ACTION actSetupMode:
//***************************************************************
// Implements a jogging based on velocity mode
// Implements homing depending on the axis type
//   Virtual axis: move absolute to 360 degrees
//   Real axis: depending on parameter S-0-0277 ModeHoming or SetAbsRef
//***************************************************************
// Do nothing, when not enabled... 
IF SetupMode.Enable = TRUE THEN
  // Positive edge of Enable ?
  IF NOT bLatchSetupModeEnable THEN
		// SetupMode is only allowed when in ModeAb or ModeAH 
		IF( (AdminCtrlExt._OpMode.en=ModeAH) OR (AdminCtrlExt._OpMode.en=ModeAb) ) THEN
      // store original values 
      rOriVel          := VelModeCtrlExt.Velocity;
      rOriAccel        := VelModeCtrlExt.Acceleration;
      rOriDecel        := AdminCtrlExt.StopDeceleration;  // Defdb00116851 / Defdb00116875  
      rOriPos          := PosModeCtrlExt.Position;
      rOriVelPos       := PosModeCtrlExt.Velocity;
      rOriAccelPos     := PosModeCtrlExt.Acceleration;
      rOriDecelPos     := PosModeCtrlExt.Deceleration;
      enOriAxisMode    := AdminCtrlExt._OpMode.en;
  	  bOriValuesStored := TRUE;
      // activate mode AH *)
      AdminCtrlExt._OpMode.en := ModeAH;
  	  enMyActAxisMode 	      := ModeAH;
  	  uiHomingState 	      := STATE_HOMING_START;
  	  //SetupModeAck.EnableAck  := TRUE; // Acknowledge SetupMode
    ELSE
      // actual not allowed to activate SetupMode
      SUPER^.mSetError( Error      := TRUE, 
                        ErrorID    := RESOURCE_ERROR, 
             	        ErrorIdent := SETUPMODE_OPMODE_ERR);
  	  bOriValuesStored:= FALSE;
    END_IF  
  END_IF // IF NOT bLatchSetupModeEnable THEN
  
  // Check if someone did overwrite our OpMode command?
  IF( (AdminCtrlExt._OpMode.en <> enMyActAxisMode) AND (SetupModeAck.EnableAck = TRUE) ) THEN
    SetupModeAck.EnableAck := FALSE; // remove acknowledge SetupMode
	
  ELSIF SetupMode.Enable = TRUE THEN
  
    //***************************************************************
    // Jogging
    //***************************************************************
    // Jog positive direction 
    IF SetupMode.JogPlus AND NOT SetupMode.JogMinus THEN
      VelModeCtrlExt.Acceleration	:= SetupMode.Accel;
      AdminCtrlExt.StopDeceleration	:= SetupMode.Accel;  // Defdb00116851 / Defdb00116875
      VelModeCtrlExt.Velocity := SetupMode.Vel;
	  AdminCtrlExt._OpMode.en := ModeVel; 
      enMyActAxisMode := ModeVel; 
    	// Jog negative direction 
    ELSIF SetupMode.JogMinus AND NOT SetupMode.JogPlus THEN
      VelModeCtrlExt.Acceleration	:= SetupMode.Accel;
      AdminCtrlExt.StopDeceleration	:= SetupMode.Accel;  // Defdb00116851 / Defdb00116875
      VelModeCtrlExt.Velocity := -SetupMode.Vel;
  	AdminCtrlExt._OpMode.en := ModeVel;  
  	enMyActAxisMode         := ModeVel;
    ELSIF AdminCtrlExt._OpMode.en = ModeVel THEN
      // switch back when coming from Jog (do not disturb homing)
  	AdminCtrlExt._OpMode.en := ModeAH;
  	enMyActAxisMode         := ModeAH;
    END_IF

    //***************************************************************
    // Implements homing depending on the axis type
    // Virtual axis: move absolute to 360 degrees
    // Real axis with closed loop: depending on parameter S-0-0277 ModeHoming or SetAbsRef
    //***************************************************************
  (* Parameter S277 Bit7/6: only read)
				
		7/6	absolute encoder
		x0: absolute encoder not possible (Bit 7 not in use)
		01: absolute encoder is active)
		11: absolute encoder is possible but deactivated *)

    CASE uiHomingState OF
  
    STATE_HOMING_START:		
        // #####################################################################  
      	IF AdminStatusExt.AxisFeatures.OPMODE_POS = FALSE THEN
          uiHomingState := STATE_HOMING_NOT_POSSIBLE; // can not be homed, e.g. open loop
        ELSIF AdminStatusExt.AxisFeatures.REAL_AXIS = TRUE THEN
					uiHomingState := STATE_HOMING_READ_S277;   // continue with read S-0-0277
      	ELSIF AdminStatusExt.AxisFeatures.VIRTUAL_AXIS = TRUE OR AdminStatusExt.AxisFeatures.CONTROLLER_AXIS = TRUE THEN
					uiHomingState := STATE_HOMING_VIRT_AXIS;   // continue with homing virtual axis
      	ELSE 
      	  // undefined axis type
   	  	  SUPER^.mSetError( Error      := TRUE, 
       		                  ErrorID    := RESOURCE_ERROR, 
           		              ErrorIdent := HOMING_CONFIGURATION_ERR);
   	  	  uiHomingState := STATE_HOMING_ERROR;   // continue with error
  		  END_IF
  
    STATE_HOMING_READ_S277:
        // #####################################################################  
      	// first read S-0-0277 when SetupMode is activated
	 			MB_ReadParameterS277(
    		Enable:= TRUE, 
    		ParameterNumber:= FP_S_0_0277, 
    		Axis:= AdminCtrlExt.Axis );
   		  IF MB_ReadParameterS277.Done = TRUE THEN
					// store Value   
					diParameterS277 := MB_ReadParameterS277.Value;
					IF 	(diParameterS277.6 AND NOT diParameterS277.7) OR diParameterS277.8 THEN
		    	  // absolute encoder
						bAbsoluteEncoder := TRUE;
        	  uiHomingState := STATE_HOMING_ABS_REAL_AXIS; // continue with homing an absolute real axis
					ELSE
		    	  // incremental encoder
						bAbsoluteEncoder := FALSE;
        	  uiHomingState := STATE_HOMING_INC_REAL_AXIS; // continue with homing an incremental real axis
					END_IF
					// RESET FB  
    		MB_ReadParameterS277(
       		Enable:= FALSE, 
      		ParameterNumber:= FP_S_0_0277, 
      		Axis:= AdminCtrlExt.Axis );
      	ELSIF MB_ReadParameterS277.Error = TRUE THEN
    		  SUPER^.mSetError( Error      := TRUE, 
                            ErrorID    := MB_ReadParameterS277.ErrorID, 
                            ErrorIdent := MB_ReadParameterS277.ErrorIdent);
					// RESET FB  
    		  MB_ReadParameterS277(
       		  Enable:= FALSE, 
      		  ParameterNumber:= FP_S_0_0277, 
      		  Axis:= AdminCtrlExt.Axis );
        	  uiHomingState := STATE_HOMING_ERROR;   // continue with error
  		  END_IF	// end of 'IF MB_ReadParameterS277.Done = TRUE THEN'		  
	
    STATE_HOMING_ABS_REAL_AXIS:
        // ##################################################################### 
				SetupModeAck.EnableAck  := TRUE; // Acknowledge SetupMode 
    		// Homing for Real-Axis with absolute encoder
      	IF (SetupMode.Homing = TRUE) AND (bHomingOld = FALSE) THEN
       		// Set reference with absolute encoder
       		AdminCtrlExt._OpMode.en := ModeAB;
    			enMyActAxisMode         := ModeAB;
				// wait for Homing finished
      	ELSIF  AdminStatusExt.AbsRefCmdStatus = MB_SERCOS_DATA_END_OK THEN
					// command finished GOOD
					SetupModeAck.HomingAck := TRUE;
					uiHomingState := STATE_HOMING_FINISHED;
					IF SetupMode.Homing = FALSE THEN
		  		  // Input was removed. Switch back to ModeAH. HomingAck stays active for one cycle... 	
		  		  bHomingRemovedBeforeFinished := TRUE;	
					END_IF	
        // Note: problems with IndraDrive Cs. It takes time to switch to AB and the 
        // C0304 "command not allowed in AF" can happen so wait for PowerOff before 
        // setting the command set absolute reference
      	ELSIF (SetupMode.Homing = TRUE) AND 
              (AxisData[AdminCtrlExt.Axis.AxisNo].Axis_Power = FALSE) THEN
       		AdminCtrlExt.SetAbsRef := TRUE;
				ELSIF ( (AdminStatusExt.AbsRefCmdStatus = MB_SERCOS_DATA_INTERRUPTED) OR	
	    	        (AdminStatusExt.AbsRefCmdStatus = MB_SERCOS_DATA_BREAK_ERROR) OR
								(AdminStatusExt.AbsRefCmdStatus = MB_SERCOS_DATA_DATUM_FAULT)    ) THEN
					// command finished BAD
					SetupModeAck.HomingAck := FALSE;
					uiHomingState := STATE_HOMING_FINISHED;
					IF SetupMode.Homing = FALSE THEN
		  		// Input was removed. Switch back to ModeAH. 	
		  		bHomingRemovedBeforeFinished := TRUE;	
					END_IF
        END_IF // end of 'IF (SetupMode.Homing = TRUE) AND (bHomingOld = FALSE) THEN'

    STATE_HOMING_INC_REAL_AXIS:
        // #####################################################################
				SetupModeAck.EnableAck  := TRUE; // Acknowledge SetupMode
    		// Homing for Real-Axis with incremental encoder
      	IF (SetupMode.Homing = TRUE) AND (bHomingOld = FALSE) THEN
       		// Set reference with incremental encoder
       		AdminCtrlExt._OpMode.en := ModeHoming;
    			enMyActAxisMode         := ModeHoming;
      	ELSIF AdminStatusExt.CmdDone THEN
					// wait for Homing finished
					// Homing finished GOOD
					SetupModeAck.HomingAck := TRUE;
					uiHomingState := STATE_HOMING_FINISHED;
					IF SetupMode.Homing = FALSE THEN
		  		// Input was removed. Switch back to ModeAH. HomingAck stays active for one cycle... 	
		  		bHomingRemovedBeforeFinished := TRUE;	
					END_IF
      	ELSIF  DiagStatusExt.Error = TRUE AND SetupMode.Homing = FALSE THEN
					// wait for Homing finished BAD. Stay here untill the Homing is removed
					SetupModeAck.HomingAck := FALSE;
					uiHomingState := STATE_HOMING_FINISHED;
  	    // Input was removed. Switch back to ModeAH. 	
					bHomingRemovedBeforeFinished := TRUE;	
      	END_IF // end of 'IF (SetupMode.Homing = TRUE) AND (bHomingOld = FALSE) THEN'		
   
    STATE_HOMING_VIRT_AXIS:
      // #####################################################################  
			SetupModeAck.EnableAck  := TRUE; // Acknowledge SetupMode
    	// Homing for Virtual-Axis -> Move abs to position 0
      	IF (SetupMode.Homing = TRUE) AND (bHomingOld = FALSE) THEN
					// rising edge on Homing  
    			// Homing for Virtual-Axis: Move to position 0 degrees
					// use SetupMode.Vel and .Accel 
          //PosModeCtrlExt.Velocity 	:= SetupMode.Vel;
          //PosModeCtrlExt.Acceleration := SetupMode.Accel;
          //PosModeCtrlExt.Deceleration := SetupMode.Accel;
					// or set vel and acc to the maximum values 
          PosModeCtrlExt.Velocity 	:= DV_Axis[AdminCtrlExt.Axis.AxisNo].A_0_0032; // or A-0-0033?
          PosModeCtrlExt.Acceleration := DV_Axis[AdminCtrlExt.Axis.AxisNo].A_0_0034-0.001; // - 0,001 to avoid warning
          PosModeCtrlExt.Deceleration := PosModeCtrlExt.Acceleration;
	    	  PosModeCtrlExt.Position 	:= 0.0; 
					AdminCtrlExt._OpMode.en := ModePosAbs;
					enMyActAxisMode         := ModePosAbs;
      	ELSIF  AdminStatusExt.CmdDone AND AdminStatusExt.MODE_POS_ABS THEN
					// wait for Homing finished GOOD
					SetupModeAck.HomingAck := TRUE;
					uiHomingState := STATE_HOMING_FINISHED;
					IF SetupMode.Homing = FALSE THEN
		  		// Input was removed. Switch back to ModeAH. HomingAck stays active for one cycle... 	
		  		bHomingRemovedBeforeFinished := TRUE;	
          END_IF
      	ELSIF  DiagStatusExt.Error = TRUE AND SetupMode.Homing = FALSE THEN
					// wait for Homing finished BAD. Stay here untill the Homing is removed
					SetupModeAck.HomingAck := FALSE;
					uiHomingState := STATE_HOMING_FINISHED;
  	      // Input was removed. Switch back to ModeAH. 	
					bHomingRemovedBeforeFinished := TRUE;	
      	END_IF // end of 'IF (SetupMode.Homing = TRUE) AND (bHomingOld = FALSE) THEN'		
	
  STATE_HOMING_FINISHED:	
        // #####################################################################  
      	IF( ((SetupMode.Homing = FALSE) AND (bHomingOld = TRUE)) OR 
            (bHomingRemovedBeforeFinished = TRUE)                   ) THEN
					// falling edge on Homing or Homing removed before finished, reset to previous settings   
					AdminCtrlExt.SetAbsRef := FALSE;
        	AdminCtrlExt._OpMode.en := ModeAH;
					enMyActAxisMode         := ModeAH;
					// remove Acknowledge
					SetupModeAck.HomingAck := FALSE;
					bHomingRemovedBeforeFinished := FALSE;
					// wait for the next rising edge on Homing input
					IF AdminStatusExt.AxisFeatures.REAL_AXIS = TRUE THEN
						IF bAbsoluteEncoder = TRUE THEN
		      	  // absolute encoder
			  		  uiHomingState := STATE_HOMING_ABS_REAL_AXIS; // continue with homing an absolute real axis
		    	  ELSE
		      	  // incremental encoder
              uiHomingState := STATE_HOMING_INC_REAL_AXIS; // continue with homing an incremental real axis
						END_IF	
          ELSE 
		   		  uiHomingState := STATE_HOMING_VIRT_AXIS;   // continue with homing virtual axis
          END_IF
				END_IF	

    STATE_HOMING_NOT_POSSIBLE:
		  ; // nothing to do
      
    STATE_HOMING_ERROR:
      // #####################################################################  
  		IF AdminCtrlExt.ClearError THEN
     		uiHomingState := STATE_HOMING_START;   // try a new start
  		END_IF	
	   

    ELSE 
        // #####################################################################  
   			// invalid state
   			SUPER^.mSetError( Error      := TRUE, 
       		              ErrorID    := STATE_MACHINE_ERROR, 
          	 	          ErrorIdent := HOMING_STATE_MACHINE_ERR);
   			uiHomingState := STATE_HOMING_ERROR;   // continue with error
	
    END_CASE // end of 'CASE uiHomingState OF'
  END_IF  // end of 'ELSIF SetupModeAck.SetupModeAck = TRUE THEN'
 
// Negative edge of Enable ? AND SetupMode was not aborted by assigning a new OpMode  
ELSIF bLatchSetupModeEnable AND bOriValuesStored = TRUE AND SetupModeAck.EnableAck = TRUE THEN
  // restore original values 
  VelModeCtrlExt.Velocity       := rOriVel;
  VelModeCtrlExt.Acceleration   := rOriAccel;
  AdminCtrlExt.StopDeceleration := rOriDecel;  // Defdb00116851 / Defdb00116875
  PosModeCtrlExt.Position       := rOriPos;
  PosModeCtrlExt.Velocity       := rOriVelPos;
  PosModeCtrlExt.Acceleration   := rOriAccelPos;
  PosModeCtrlExt.Deceleration   := rOriDecelPos;
  AdminCtrlExt._OpMode.en       := enOriAxisMode;
  bOriValuesStored              := FALSE;
  SetupModeAck.EnableAck        := FALSE; // remove acknowledge SetupMode
END_IF // SetupMode.Enable = TRUE

bLatchSetupModeEnable := SetupMode.Enable;
bHomingOld            := SetupMode.Homing;
END_ACTION

ACTION actSyncAccVel:
// Implements writing the Sync-Acceleration into parameter A-0-2791
// and writing the Sync-Velocity into parameter A-0-2790
// ####################################################
// Check if we are in bb. Otherwise we get errors.
// Do this only when sync is supported and the parameters are available.
// Distribute the load with using the axis address
IF AxisData[AdminCtrlExt.Axis.AxisNo].Axis_OperationMode = TRUE    AND 
   AdminStatusExt.AxisFeatures.OPMODE_SYNC = TRUE                   AND 
   (udiCycleCntInP4 > DINT_TO_UDINT(2 * AdminCtrlExt.Axis.AxisNo))     THEN 
  // write SyncAcceleration when changed 
  IF SyncModeCtrlExt.SyncAcceleration <> rLastSyncAcc THEN
    // start transmission 
    SyncModeStatusExt.SyncAccelerationDone := FALSE;
    bExecWrSyncAcc := TRUE;
  END_IF
  IF fbWrSyncAcc.Done = TRUE THEN 
    // finished GOOD transmission 
    SyncModeStatusExt.SyncAccelerationDone := TRUE;
    bExecWrSyncAcc := FALSE;
    // remember old value 
    rLastSyncAcc := SyncModeCtrlExt.SyncAcceleration;
  ELSIF fbWrSyncAcc.Error = TRUE THEN  
    // finished BAD transmission 
    bExecWrSyncAcc := FALSE;
    SUPER^.mSetError( Error      := TRUE, 
                      ErrorID    := fbWrSyncAcc.ErrorID, 
                      ErrorIdent := fbWrSyncAcc.ErrorIdent);
    // remember old value, to not write cyclically bad values 
    rLastSyncAcc := SyncModeCtrlExt.SyncAcceleration;
  END_IF  
  // call FB 
  fbWrSyncAcc(
	Execute:= bExecWrSyncAcc, 
	ParameterNumber:= FP_A_0_2791, 
	Value:= SyncModeCtrlExt.SyncAcceleration, 
	Axis:= AdminCtrlExt.Axis );	
	
  // ####################################################
  // write SyncVelocity when changed 
  IF SyncModeCtrlExt.SyncVelocity <> rLastSyncVel THEN
    // start transmission 
    SyncModeStatusExt.SyncVelocityDone := FALSE;
    bExecWrSyncVel := TRUE;
  END_IF
  IF fbWrSyncVel.Done = TRUE THEN 
    // finished GOOD transmission 
    SyncModeStatusExt.SyncVelocityDone := TRUE;
    bExecWrSyncVel := FALSE;
    // remember old value 
    rLastSyncVel := SyncModeCtrlExt.SyncVelocity;
  ELSIF fbWrSyncVel.Error = TRUE THEN  
    // finished BAD transmission 
    bExecWrSyncVel := FALSE;
    SUPER^.mSetError( Error      := TRUE, 
                      ErrorID    := fbWrSyncVel.ErrorID, 
                      ErrorIdent := fbWrSyncVel.ErrorIdent);
    // remember old value, to not write cyclically bad values 
    rLastSyncVel := SyncModeCtrlExt.SyncVelocity;
  END_IF  
  // call FB 
  fbWrSyncVel(
	Execute:= bExecWrSyncVel, 
	ParameterNumber:= FP_A_0_2790, 
	Value:= SyncModeCtrlExt.SyncVelocity, 
	Axis:= AdminCtrlExt.Axis );	
ELSE
  // reset FBs when not in bb 
  fbWrSyncAcc( Execute:= FALSE,	Axis:= AdminCtrlExt.Axis );	
  fbWrSyncVel( Execute:= FALSE,	Axis:= AdminCtrlExt.Axis );	
END_IF
END_ACTION

ACTION actCopyAxisData_HMI:
// copy AxisData status informations to AxisData_HMI structure to transmit to HMI

AxisData_HMI.dwMotionProfileStatusBits_i    	:=	AxisData[AdminCtrlExt.Axis.AxisNo].dwMotionProfileStatusBits_i;	
AxisData_HMI.FlexProfil_Sync                    :=  AxisData[AdminCtrlExt.Axis.AxisNo].FlexProfil_Sync;                 
AxisData_HMI.FlexProfil_Active                  :=  AxisData[AdminCtrlExt.Axis.AxisNo].FlexProfil_Active;               
AxisData_HMI.FlexProfil_WaitForSwitching        :=  AxisData[AdminCtrlExt.Axis.AxisNo].FlexProfil_WaitForSwitching;     
AxisData_HMI.FlexProfil_Set0_Checked            :=  AxisData[AdminCtrlExt.Axis.AxisNo].FlexProfil_Set0_Checked;         
AxisData_HMI.FlexProfil_Set0_Ok                 :=  AxisData[AdminCtrlExt.Axis.AxisNo].FlexProfil_Set0_Ok;              
AxisData_HMI.FlexProfil_Set1_Checked            :=  AxisData[AdminCtrlExt.Axis.AxisNo].FlexProfil_Set1_Checked;         
AxisData_HMI.FlexProfil_Set1_Ok                 :=  AxisData[AdminCtrlExt.Axis.AxisNo].FlexProfil_Set1_Ok;              
AxisData_HMI.FlexProfil_Set2_Checked            :=  AxisData[AdminCtrlExt.Axis.AxisNo].FlexProfil_Set2_Checked;         
AxisData_HMI.FlexProfil_Set2_Ok                 :=  AxisData[AdminCtrlExt.Axis.AxisNo].FlexProfil_Set2_Ok;              
AxisData_HMI.FlexProfil_Set3_Checked            :=  AxisData[AdminCtrlExt.Axis.AxisNo].FlexProfil_Set3_Checked;         
AxisData_HMI.FlexProfil_Set3_Ok                 :=  AxisData[AdminCtrlExt.Axis.AxisNo].FlexProfil_Set3_Ok;              
AxisData_HMI.FlexProfil_EvtSet0_Checked         :=  AxisData[AdminCtrlExt.Axis.AxisNo].FlexProfil_EvtSet0_Checked;      
AxisData_HMI.FlexProfil_EvtSet0_Ok              :=  AxisData[AdminCtrlExt.Axis.AxisNo].FlexProfil_EvtSet0_Ok;           
AxisData_HMI.FlexProfil_EvtSet1_Checked         :=  AxisData[AdminCtrlExt.Axis.AxisNo].FlexProfil_EvtSet1_Checked;      
AxisData_HMI.FlexProfil_EvtSet1_Ok              :=  AxisData[AdminCtrlExt.Axis.AxisNo].FlexProfil_EvtSet1_Ok;           
AxisData_HMI.FlexProfil_EvtSet2_Checked         :=  AxisData[AdminCtrlExt.Axis.AxisNo].FlexProfil_EvtSet2_Checked;      
AxisData_HMI.FlexProfil_EvtSet2_Ok              :=  AxisData[AdminCtrlExt.Axis.AxisNo].FlexProfil_EvtSet2_Ok;           
AxisData_HMI.FlexProfil_EvtSet3_Checked         :=  AxisData[AdminCtrlExt.Axis.AxisNo].FlexProfil_EvtSet3_Checked;      
AxisData_HMI.FlexProfil_EvtSet3_Ok              :=  AxisData[AdminCtrlExt.Axis.AxisNo].FlexProfil_EvtSet3_Ok;           
AxisData_HMI.dwFlexProfileEventStatusBits_i     :=  AxisData[AdminCtrlExt.Axis.AxisNo].dwFlexProfileEventStatusBits_i; 
AxisData_HMI.Axis_CamTab_0                      :=  AxisData[AdminCtrlExt.Axis.AxisNo].Axis_CamTab_0;                   
AxisData_HMI.Axis_CamTab_1                      :=  AxisData[AdminCtrlExt.Axis.AxisNo].Axis_CamTab_1;                   
AxisData_HMI.Axis_CamTab_2                      :=  AxisData[AdminCtrlExt.Axis.AxisNo].Axis_CamTab_2;                   
AxisData_HMI.Axis_CamSwitching                  :=  AxisData[AdminCtrlExt.Axis.AxisNo].Axis_CamSwitching;               
AxisData_HMI.Axis_InVelocity                    :=  AxisData[AdminCtrlExt.Axis.AxisNo].Axis_InVelocity;                 
AxisData_HMI.Axis_Standstill                    :=  AxisData[AdminCtrlExt.Axis.AxisNo].Axis_Standstill;                 
AxisData_HMI.Axis_InPosition                    :=  AxisData[AdminCtrlExt.Axis.AxisNo].Axis_InPosition;      
AxisData_HMI.Axis_InSynchron                    :=  AxisData[AdminCtrlExt.Axis.AxisNo].Axis_InSynchron;                 
AxisData_HMI.Axis_Warning                       :=  AxisData[AdminCtrlExt.Axis.AxisNo].Axis_Warning;                    
AxisData_HMI.Axis_Error                         :=  AxisData[AdminCtrlExt.Axis.AxisNo].Axis_Error;                      
AxisData_HMI.Axis_Homed                         :=  AxisData[AdminCtrlExt.Axis.AxisNo].Axis_Homed;                      
AxisData_HMI.Axis_InTorque                      :=  AxisData[AdminCtrlExt.Axis.AxisNo].Axis_InTorque;                   
AxisData_HMI.Axis_OperationMode                 :=  AxisData[AdminCtrlExt.Axis.AxisNo].Axis_OperationMode;              
AxisData_HMI.Axis_Inbb                          :=  AxisData[AdminCtrlExt.Axis.AxisNo].Axis_Inbb;                       
AxisData_HMI.Axis_InAb                          :=  AxisData[AdminCtrlExt.Axis.AxisNo].Axis_InAb;                       
AxisData_HMI.Axis_Power                         :=  AxisData[AdminCtrlExt.Axis.AxisNo].Axis_Power;                      
AxisData_HMI.Axis_CmdActive                     :=  AxisData[AdminCtrlExt.Axis.AxisNo].Axis_CmdActive;                  
AxisData_HMI.Axis_ErrInProgress                 :=  AxisData[AdminCtrlExt.Axis.AxisNo].Axis_ErrInProgress;              
AxisData_HMI.Axis_CyclicPosChannelOpen          :=  AxisData[AdminCtrlExt.Axis.AxisNo].Axis_CyclicPosChannelOpen;       
AxisData_HMI.Axis_InMasterPhaseOffset           :=  AxisData[AdminCtrlExt.Axis.AxisNo].Axis_InMasterPhaseOffset;        
AxisData_HMI.Axis_CyclicTrqChannelOpen          :=  AxisData[AdminCtrlExt.Axis.AxisNo].Axis_CyclicTrqChannelOpen;       
AxisData_HMI.Axis_CyclicVelChannelOpen          :=  AxisData[AdminCtrlExt.Axis.AxisNo].Axis_CyclicVelChannelOpen;       
AxisData_HMI.Axis_CyclicAnaChannelOpen          :=  AxisData[AdminCtrlExt.Axis.AxisNo].Axis_CyclicAnaChannelOpen;       
AxisData_HMI.ErrorStop                          :=  AxisData[AdminCtrlExt.Axis.AxisNo].ErrorStop;                       
AxisData_HMI.Stopping                           :=  AxisData[AdminCtrlExt.Axis.AxisNo].Stopping;                        
AxisData_HMI.Homing                             :=  AxisData[AdminCtrlExt.Axis.AxisNo].Homing;                          
AxisData_HMI.PowerOn                            :=  AxisData[AdminCtrlExt.Axis.AxisNo].PowerOn;                         
AxisData_HMI.DiscreteMotion                     :=  AxisData[AdminCtrlExt.Axis.AxisNo].DiscreteMotion;                  
AxisData_HMI.ContinuousMotion                   :=  AxisData[AdminCtrlExt.Axis.AxisNo].ContinuousMotion;                
AxisData_HMI.SynchronizedMotion                 :=  AxisData[AdminCtrlExt.Axis.AxisNo].SynchronizedMotion;              
AxisData_HMI.Standstill                         :=  AxisData[AdminCtrlExt.Axis.AxisNo].Standstill;                      
AxisData_HMI.CoordinatedMotion                  :=  AxisData[AdminCtrlExt.Axis.AxisNo].CoordinatedMotion;               
AxisData_HMI.ControlledMotion                   :=  AxisData[AdminCtrlExt.Axis.AxisNo].ControlledMotion;                
AxisData_HMI.dwAxisCondition_i                  :=  AxisData[AdminCtrlExt.Axis.AxisNo].dwAxisCondition_i;               
AxisData_HMI.rActualPosition_i                  :=  AxisData[AdminCtrlExt.Axis.AxisNo].rActualPosition_i;               
AxisData_HMI.rActualVelocity_i                  :=  AxisData[AdminCtrlExt.Axis.AxisNo].rActualVelocity_i;               
AxisData_HMI.rActualTorqueForce_i               :=  AxisData[AdminCtrlExt.Axis.AxisNo].rActualTorqueForce_i;            
AxisData_HMI.wUserActualDataBitA_i              :=  AxisData[AdminCtrlExt.Axis.AxisNo].wUserActualDataBitA_i;          
AxisData_HMI.wUserActualDataBitB_i              :=  AxisData[AdminCtrlExt.Axis.AxisNo].wUserActualDataBitB_i;          
AxisData_HMI.wUserActualDataBitC_i              :=  AxisData[AdminCtrlExt.Axis.AxisNo].wUserActualDataBitC_i;          
AxisData_HMI.wUserActualDataBitD_i              :=  AxisData[AdminCtrlExt.Axis.AxisNo].wUserActualDataBitD_i;          
AxisData_HMI.dwUserActualDataA_i                :=  AxisData[AdminCtrlExt.Axis.AxisNo].dwUserActualDataA_i;             
AxisData_HMI.dwUserActualDataB_i                :=  AxisData[AdminCtrlExt.Axis.AxisNo].dwUserActualDataB_i;             
AxisData_HMI.dwUserActualDataC_i                :=  AxisData[AdminCtrlExt.Axis.AxisNo].dwUserActualDataC_i;             
AxisData_HMI.dwUserActualDataD_i                :=  AxisData[AdminCtrlExt.Axis.AxisNo].dwUserActualDataD_i;             
AxisData_HMI.dwUserActualDataE_i                :=  AxisData[AdminCtrlExt.Axis.AxisNo].dwUserActualDataE_i;             
AxisData_HMI.dwUserActualDataF_i                :=  AxisData[AdminCtrlExt.Axis.AxisNo].dwUserActualDataF_i;
END_ACTION

METHOD mInitExtension
VAR_INPUT
	index: UINT;
END_VAR
VAR
END_VAR
SUPER^.mInitExtension(index);

IF NOT bFirstInit THEN
	// User: Assigment of user defined axis interface inputs
	SetupMode  REF= arAxisCtrl_gb[index].SetupMode;
	
	// User: Assigment of user defined axis interface outputs
	SetupModeAck REF= arAxisStatus_gb[index].SetupMode;
	AxisData_HMI REF= arAxisStatus_gb[index].AxisData_HMI;
	
	// =================================================================
	// Do not touch the following lines
	// =================================================================
	
	// Set the references for the AxisInterface FB 
	AdminCtrlExt   	REF= arAxisCtrl_gb[index].Admin;
	PosModeCtrlExt    REF= arAxisCtrl_gb[index].PosMode;
	VelModeCtrlExt    REF= arAxisCtrl_gb[index].VelMode;
	SyncModeCtrlExt   REF= arAxisCtrl_gb[index].SyncMode;
	AdminStatusExt    REF= arAxisStatus_gb[index].Admin;
	DiagStatusExt     REF= arAxisStatus_gb[index].Diag;
	PosStatusExt   	REF= arAxisStatus_gb[index].PosMode;
	VelStatusExt      REF= arAxisStatus_gb[index].VelMode;
	SyncModeStatusExt REF= arAxisStatus_gb[index].SyncMode;
	// System: assign references of axis interface refresh FB
	AdminCtrl 				REF= arAxisCtrl_gb[index].Admin;
	PosModeCtrl 			REF= arAxisCtrl_gb[index].PosMode;
	VelModeCtrl 			REF= arAxisCtrl_gb[index].VelMode;
	SyncModeCtrl 			REF= arAxisCtrl_gb[index].SyncMode;
	AdminStatus 			REF= arAxisStatus_gb[index].Admin;
	DiagStatus 				REF= arAxisStatus_gb[index].Diag;
	PosStatus 				REF= arAxisStatus_gb[index].PosMode;
	VelStatus 				REF= arAxisStatus_gb[index].VelMode;
	SyncModeStatus 		REF= arAxisStatus_gb[index].SyncMode;
END_IF
END_METHOD

END_FUNCTION_BLOCK

// IndraMotionMlc1/Application/Utilities/InitAxis
PROGRAM InitAxis
VAR
	index:INT;
END_VAR
VAR_INPUT
	
	arAxisPointer: POINTER TO ARRAY[1..20] OF AXIS_REF;
	uiNUM_FLEXO_F: UINT;
	
END_VAR

FOR index:=1 TO uiNUM_FLEXO_F BY 1 DO
		arAxisCtrl_gb[arAxisPointer^[index].AxisNo].SyncMode.InputRevolution := 1000;
		arAxisCtrl_gb[arAxisPointer^[index].AxisNo].SyncMode.OutputRevolution := 1000;
		arAxisCtrl_gb[arAxisPointer^[index].AxisNo].SyncMode.Master:=VMA_FT1;
		arAxisCtrl_gb[arAxisPointer^[index].AxisNo].SyncMode.StartMode:=RELATIVE;
		arAxisCtrl_gb[arAxisPointer^[index].AxisNo].SyncMode.SyncAcceleration:=1.0;
		arAxisCtrl_gb[arAxisPointer^[index].AxisNo].SyncMode.PhaseOffsetAcc:=1.0;
		arAxisCtrl_gb[arAxisPointer^[index].AxisNo].SyncMode.SyncDirection:=SHORTEST_WAY;
		arAxisCtrl_gb[arAxisPointer^[index].AxisNo].SyncMode.SyncVelocity:=5.0;
	END_FOR

END_PROGRAM

// IndraMotionMlc1/Application/STATE_MACHINE/Winder
PROGRAM Winder
VAR_INPUT
	arAxisPointer: POINTER TO ARRAY[1..20] OF AXIS_REF;
	uiNUM_FLEXO_F: UINT;
	MACHINE_STATE_i:STATE;
	iGearValue :INT;
END_VAR
VAR_OUTPUT
	
	bRewIntrlock:BOOL;
END_VAR

//(ERROR_CHECK,SETUP_PREPARE,SETUP_WAIT,SETUP_P2,SETUP_WRITEGEAR,SETUP_WRITEGEAR_WAIT,SETUP_P4,INIT_SYNC,INIT_VERIFY,
//HOLD,RUN_PREPARE,RUN_DELAY,RUN,JOG_PREPARE,JOG_DELAY,JOG,JOG_WAIT,ERROR);



IF MACHINE_STATE_i = HOLD THEN
	arAxisCtrl_gb[arAxisPointer^[1].AxisNo].Admin._OpMode.en:=ModeSyncVel;
ELSIF MACHINE_STATE_i = ERROR THEN
	arAxisCtrl_gb[arAxisPointer^[1].AxisNo].Admin._OpMode.en:=ModeAB;
END_IF

END_PROGRAM

// IndraMotionMlc1/Application/REF_SPEED/SetVmaSpeed
PROGRAM SetVmaSpeed
VAR
	rRunVmaSpeedRpm:REAL;
	rRunVmaSpeedInch:REAL;
	rJogVmaSpeedRpm:REAL;
	rJogVmaSpeedInch:REAL;
END_VAR
VAR_INPUT
	arAxisPointer: POINTER TO ARRAY[1..20] OF AXIS_REF;
	uiNUM_FLEXO_F: UINT;
	rFormat:REAL;
	rRunSpeedDemandFPM:REAL; //(0 to 6000 in/m)
	rJogSpeedDemandFPM:REAL; //(0 to 6000 in/m)
	uiState:STATE;
END_VAR

//SetSpeedFPM (0 to 6000 inpm)
//Format 1 to 20 inches

//SetVMASpeed(Format, SetSpeedFPM)
//AdjustElectronicRatio(uiNUM_FLEXO)

//***********************	
//CALCULATE VMA SPEED !!!
//***********************		
//12 inches format  RUN DEMAND
//Example for a apeed demand of 100 rpm
//and a 8 inch format..
//we will get a VMA at (12/8)*100 rpm = 150 rpm
arAxisCtrl_gb[VMA_FT1.AxisNo].VelMode.Acceleration := 1.0;
arAxisCtrl_gb[VMA_FT1.AxisNo].VelMode.Deceleration := 1.0;

rRunVmaSpeedInch 	:= (rRunSpeedDemandFPM*12.0); //in inches
rRunVmaSpeedRpm		:=  rRunVmaSpeedInch/rFormat;

//12 inches format  JOG DEMAND
rJogVmaSpeedInch 	:= (rJogSpeedDemandFPM*12.0); //in inches
rJogVmaSpeedRpm		:=  rJogVmaSpeedInch/rFormat;	




IF uiState = RUN THEN

	arAxisCtrl_gb[VMA_FT1.AxisNo].VelMode.Velocity := rRunVmaSpeedRpm;

ELSIF uiState = JOG THEN
	arAxisCtrl_gb[VMA_FT1.AxisNo].VelMode.Velocity := rJogVmaSpeedRpm;
ELSE
	arAxisCtrl_gb[VMA_FT1.AxisNo].VelMode.Velocity := 0.0;
END_IF

END_PROGRAM

// IndraMotionMlc1/Application/FormatC
PROGRAM FormatC
VAR_IN_OUT
	bExecute:BOOL;
END_VAR
VAR
	
	fbWriteGearInL: MB_WriteLintParameter;
	arliNewFormat: ARRAY[1..10] OF LINT;
	arfbWriteGearInL: ARRAY[1..10] OF MB_WriteLintParameter;
	index:UINT;
	
	MB_writepar: MB_WriteParameter;
	WriteGear: ARRAY[1..20] OF MB_WriteParameter;
	bWriteExec: ARRAY[1..20] OF BOOL;
	uiState:UINT;
	bWriteIsDone:BOOL;
END_VAR
VAR_INPUT
	arAxisPointer: POINTER TO ARRAY[1..20] OF AXIS_REF;
	uiNUM_FLEXO_F: UINT;
	MACHINE_STATE_i:STATE;
	iGearValue :INT;
END_VAR
VAR_OUTPUT
	bSetupDone_i:BOOL;
END_VAR

IF MACHINE_STATE_i = SETUP_WRITEGEAR_WAIT THEN
	IF (iGearValue > 1000)THEN

		FOR index:=1 TO uiNUM_FLEXO_F BY 1 DO
			WriteGear[index](
			Execute:=, 
			ParameterNumber:=GVL_S_Param_ID.FP_S_0_0121 , 
			Value:=iGearValue , 
			Axis:= arAxisPointer^[index], 
			Done=> , 
			Active=> , 
			Error=> , 
			ErrorID=> , 
			ErrorIdent=> );
			
			arAxisCtrl_gb[arAxisPointer^[index].AxisNo].SyncMode.OutputRevolution := INT_TO_UINT(iGearValue);
			arAxisCtrl_gb[arAxisPointer^[index].AxisNo].SyncMode.InputRevolution := 9600;
		END_FOR
	END_IF	
	CASE uiState OF 
		COMMAND:
			IF bExecute THEN
				FOR index:=1 TO uiNUM_FLEXO_F BY 1 DO	
					WriteGear[index].Execute := TRUE;
				END_FOR
					uiState := WAIT;
			END_IF
		WAIT:
			bWriteIsDone:=TRUE;
			FOR index:=1 TO uiNUM_FLEXO_F BY 1 DO	
				bWriteIsDone := bWriteIsDone AND WriteGear[index].Done;
			END_FOR
			IF bWriteIsDone THEN uiState := DONE; END_IF
		DONE:
			uiState := COMMAND;
			bExecute := FALSE;
			FOR index:=1 TO uiNUM_FLEXO_F BY 1 DO	
				WriteGear[index].Execute := FALSE;
			END_FOR
			
	END_CASE;
END_IF

END_PROGRAM

// IndraMotionMlc1/Application/MAIN_PGM/GravureState
PROGRAM GravureState
VAR
	

	bVM_Enable: BOOL;
	rVM_Acc: REAL:=10.0;
	rVM_Dec: REAL:=10.0;
	rVM_Velocity: REAL:=0.0;
	bVM_VelModeAck: BOOL;
	bVM_Standstill: BOOL;
	rVM_actVelocity: REAL;
	bSynch: BOOL;
	rFineAdjust: REAL := 0;
	fbTimerToSlowRotation: TON;
	rSlowRotationAccel: REAL := 5.0;
	rSlowRotationVel: REAL := 5.0;
	uiState: INT;

	bInit: BOOL;
	fbSynchCnt: R_TRIG;
	iSynchCnt: INT;
	
	fbWriteExpectWindows: MB_WriteExpectWindow;
	rRecordedPosition:REAL;
	
END_VAR

VAR_OUTPUT
	dwUserActualDataB_i: INT;
END_VAR

//------------------------------------------------------------------------------------------------------
//--------------------- Call all required programs --> Imc and Axis Interface Update  ------------------  
//------------------------------------------------------------------------------------------------------
TE_AxisInterfaceType01Prog();
MB_ImcInterface();

IF TE_AxisInterfaceType01Prog.InitDone=FALSE THEN
	RETURN;
END_IF


//SYNCHRONIZE VMA_TO_REALMASTER



IF NOT binit THEN 
	
	//VMA est synchronizé à l'encodeur de l'essieu principal (REAL MASTER)
	//on applique un ratio correspondant au format
	//Essieu principal est 96 dents
	//Gravure est de 132 dents
	arAxisCtrl_gb[arDrive[1].AxisNo].SyncMode.InputRevolution := 13200;
	arAxisCtrl_gb[arDrive[1].AxisNo].SyncMode.OutputRevolution := 9600;
	arAxisCtrl_gb[arDrive[1].AxisNo].SyncMode.Master:=VMA_FT;
	arAxisCtrl_gb[arDrive[1].AxisNo].SyncMode.StartMode:=RELATIVE;
	arAxisCtrl_gb[arDrive[1].AxisNo].SyncMode.SyncAcceleration:=1.0;
	arAxisCtrl_gb[arDrive[1].AxisNo].SyncMode.PhaseOffsetAcc:=1.0;
	arAxisCtrl_gb[arDrive[1].AxisNo].SyncMode.SyncDirection:=SHORTEST_WAY;
	arAxisCtrl_gb[arDrive[1].AxisNo].SyncMode.SyncVelocity:=5.0;
	uiState:=0;

ELSE


	AUTO_REGISTER();

CASE uiState OF
	
	99:
		arAxisCtrl_gb[arDrive[1].AxisNo].Admin._OpMode.en:= ModeHoming;	
		IF  arAxisStatus_gb[1].Admin.CmdDone AND AxisData[1].Axis_Homed AND AxisData[1].Axis_Standstill THEN
				uiState:= 0;	//HOMING IS DONE
		END_IF

	0: //Wait for Synch
		arAxisCtrl_gb[arDrive[1].AxisNo].Admin._OpMode.en:= ModeAB;
		IF bGravureOn_ETH_q    THEN
			uiState:=5;
		END_IF
	//3://CREEP AND FIND THE MARK ON CYLINDER
		
	
	
		
	
	5:	//Wait for Homing
		arAxisCtrl_gb[arDrive[1].AxisNo].Admin._OpMode.en:= ModeHoming;	
		IF  arAxisStatus_gb[1].Admin.CmdDone AND AxisData[1].Axis_Homed AND AxisData[1].Axis_Standstill THEN
			uiState:= 10;	//HOMING IS DONE
		END_IF
			
		IF NOT bGravureOn_ETH_q    THEN
			uiState:=0;
		END_IF
		
	10://Synch to Master
	
		arAxisCtrl_gb[arDrive[1].AxisNo].Admin._OpMode.en:= ModeSyncPhase;
		IF arAxisStatus_gb[arDrive[1].AxisNo].Admin._OpModeAck = ModeSyncPhase THEN 
			uiState:=20;
		END_IF
			
		IF (NOT bGravureOn_ETH_q)    THEN
			uiState:=0;
		END_IF
		
	20://Check for Slow Rotation Conditions
	
		IF (bGravureSlowRot_ETH_i = TRUE)	AND (bRewindPID_Out_i = FALSE) THEN
			uiState:=30;
		END_IF
		IF (NOT bGravureOn_ETH_q)    THEN
			uiState:=0;
		END_IF
	
	30:
		//rRecordedPosition := arAxisCtrl_gb[1].PosMode.Position
		rRecordedPosition := arAxisStatus_gb[arDrive[1].AxisNo].PtrAxisData^.rActualPosition_i;
		arAxisCtrl_gb[arDrive[1].AxisNo].Admin._OpMode.en:= ModeAB;
				//arAxisCtrl[Axis1.Axisno].Admin._OpMode := ModePosAbs;
		IF arAxisStatus_gb[arDrive[1].AxisNo].Admin._OpModeAck = ModeAB THEN 
			uiState:=35;
		END_IF
		IF (NOT bGravureOn_ETH_q)    THEN
			uiState:=0;
		END_IF
	//33:		//HOME THE  AXIS
			//SKIP THIS PART!!!
		//arAxisCtrl_gb[arDrive[1].AxisNo].Admin._OpMode.en:= ModeHoming;	
		//IF  arAxisStatus_gb[1].Admin.CmdDone AND AxisData[1].Axis_Homed AND AxisData[1].Axis_Standstill THEN
		//	uiState:= 35;	//HOMING IS DONE
		//END_IF
		//IF (NOT bGravureOn_ETH_q)    THEN
		//	uiState:=0;
		//END_IF
	35:// Enable Slow Rotation:
		IF bRewindPID_Out_i = FALSE THEN
			arAxisCtrl_gb[arDrive[1].AxisNo].VelMode.Acceleration:= rSlowRotationAccel;
			arAxisCtrl_gb[arDrive[1].AxisNo].VelMode.Velocity:=5.0;
			arAxisCtrl_gb[arDrive[1].AxisNo].Admin._OpMode.en:= ModeVel;
		END_IF
			
			IF arAxisStatus_gb[arDrive[1].AxisNo].Admin._OpModeAck=ModeVel THEN 
				uiState:= 40;
			END_IF
		IF (NOT bGravureOn_ETH_q)    THEN
			uiState:=0;
		END_IF
	40: // Wait For Speed Up
		
		//BACK TO SYNCHRONIZE  Hommie!!!
		IF ((bRewindPID_Out_i OR NOT bGravureSlowRot_ETH_i) AND(bGravureOn_ETH_q=TRUE))THEN
		
			uiState:= 50;
		END_IF

	
		IF (NOT bGravureOn_ETH_q)    THEN
			uiState:=0;
		END_IF
	50:
	
			arAxisCtrl_gb[arDrive[1].AxisNo].Admin._OpMode.en:= ModeAB;
		IF arAxisStatus_gb[arDrive[1].AxisNo].Admin._OpModeAck = ModeAB THEN 
			uiState:=55;
		END_IF
		IF (NOT bGravureOn_ETH_q)    THEN
			uiState:=0;
		END_IF
	55:		
			arAxisCtrl_gb[arDrive[1].AxisNo].VelMode.Velocity:=20.0;
			arAxisCtrl_gb[arDrive[1].AxisNo].PosMode.Velocity:=20.0;
			arAxisCtrl_gb[arDrive[1].AxisNo].PosMode.Position := rRecordedPosition;
			
			arAxisCtrl_gb[arDrive[1].AxisNo].Admin._OpMode.en:= ModePosAbs;
		IF arAxisStatus_gb[arDrive[1].AxisNo].Admin._OpModeAck = ModePosAbs THEN 
			uiState:=60;
		END_IF
		IF (NOT bGravureOn_ETH_q)    THEN
			uiState:=0;
		END_IF
			
	60:
			
		
		
		IF arAxisStatus_gb[arDrive[1].AxisNo].Admin._OpModeAck = ModePosAbs AND arAxisStatus_gb[1].Admin.CmdDone = TRUE THEN 
		
			IF bGravureOn_ETH_q    THEN
				uiState:=10;
			ELSE
				uiState:=0;
			END_IF
		END_IF
	
END_CASE
END_IF
bInit:=TRUE;

END_PROGRAM

// IndraMotionMlc1/Application/AUTO_REGISTER
PROGRAM AUTO_REGISTER
VAR
	
uiState_2:	UINT;


	//	bGravureRegiOn_HMI_i: BOOL;
	//	bPauseRegiOn_HMI_i: BOOL;
	//	bSetPtLckRegiCtrl_HMI_i: BOOL;
	//	bSetPtLckRegiCtrlAck_HMI_q: BOOL;
	
		uiLatchPosEdge:UINT;
	//	uiCountPosEdge_gb:UINT
	uiCountPosEdge_gb: UINT	:= 0;
	bFlag:BOOL;
	
	bOpenRegWindow:BOOL:=FALSE;
	
	bWriteExpectWindow:BOOL;
	rCheckStart: REAL;
	rCheckStop: REAL;
	uiCheckStart: UINT;
	uiCheckStop: UINT;
	
	rEffectiveStartWin:REAL;
	rEffectiveStopWin:REAL;
	uiEffectiveStartWin:UINT;
	uiEffectiveStopWin:UINT;
END_VAR


AdjustPreset();
WriteExpectWindow();


CASE uiState_2 OF
	
	0: //AUTO REGISTER IS OFF AND SYNC OFF
		bOpenRegWindow 		:= TRUE;
		uiCountPosEdge_gb:= 0;
		//bSetPtLckRegiCtrl_HMI_i := FALSE;
		bPauseRegiOn_HMI_i 			:= TRUE;
		bSetPtLckRegiCtrl_HMI_i 	:= FALSE;
		
		IF arAxisStatus_gb[Drive1.AxisNo].Admin._OpModeAck = ModeSyncPhase THEN 
			uiState_2:=10;
		END_IF
		
	10://AXIS IS SYNCHRONIZED
	
	
		IF arAxisStatus_gb[Drive1.AxisNo].Admin._OpModeAck = ModeSyncPhase THEN
			
			//STOP WRITING TO P694
			bPauseRegiOn_HMI_i 			:= TRUE;
		
			IF bGravureRegiOn_HMI_i = TRUE THEN
				
				
				//EXECUTE WRITE EXPECTATION
				rSetPointWindows_gb := 180.0;
				bWriteExpectWindow := FALSE;		
				rExpectWindowPosEdgeStart_gb :=179.99;
				rExpectWindowPosEdgeEnd_gb	:=179.99;
				bWriteExpectWindow := TRUE;
				
				//READ VALUE IN PROBE
				rEffectiveStartWin:=AxisData[Drive1.AxisNo].dwUserActualDataC_i.REAL_;
				rEffectiveStopWin:=AxisData[Drive1.AxisNo].dwUserActualDataD_i.REAL_;
				rCheckStart	:=rSetPointWindows_gb-179.99;

				IF NOT InsetterControl.fbRegiRegulate11.InOperation	AND 	
					rEffectiveStartWin =  0.01 AND rEffectiveStopWin = 359.99 THEN
					uiState_2:=30;
				END_IF	
			ELSE
				bPauseRegiOn_HMI_i 			:= TRUE;
				bWriteExpectWindow := FALSE;		//CLOSE THE WINDOW
				rExpectWindowPosEdgeStart_gb :=0.0;
				rExpectWindowPosEdgeEnd_gb	:= 0.0;
				//bWriteExpectWindow := TRUE;		
			END_IF
	
		ELSE	
			uiState_2:=0;
		END_IF
		
	
	30:
			//SEND LOCK COMMAND
			//Write a new Position Setpoint using MB_RegiSetpointLockType01
			bPauseRegiOn_HMI_i 			:= TRUE;
			bSetPtLckRegiCtrl_HMI_i 	:= TRUE;
			//IF 	 bSetPtLckRegiCtrlAck_HMI_q = TRUE AND rSetPointWindows_gb <> 0.0 THEN
			IF bSetPtLckRegiCtrlAck_HMI_q AND arAxisStatus_gb[Drive1.AxisNo].SyncMode.PhasingSlaveDone THEN		
					bSetPtLckRegiCtrl_HMI_i := FALSE;
					uiState_2:=35;
			END_IF
			
			IF 	bGravureRegiOn_HMI_i = FALSE THEN uiState_2:=0;	END_IF
			
	35:		//CLOSE THE WINDOW AROUND NEW POSITION SETPOINT
				bWriteExpectWindow := FALSE;		//CLOSE THE WINDOW
				rExpectWindowPosEdgeStart_gb :=15.0;
				rExpectWindowPosEdgeEnd_gb	:=15.0;
				bWriteExpectWindow := TRUE;
				rEffectiveStartWin:=AxisData[Drive1.AxisNo].dwUserActualDataC_i.REAL_;
				rEffectiveStopWin:=AxisData[Drive1.AxisNo].dwUserActualDataD_i.REAL_;
				rCheckStart	:=REAL_TO_UINT(rSetPointWindows_gb-15.0);
				rCheckStop	:=REAL_TO_UINT(rSetPointWindows_gb+15.0);
				
			IF uiEffectiveStartWin =  uiCheckStart AND uiEffectiveStopWin = uiCheckStop THEN
				uiState_2:=40;
			END_IF	
			IF 	bGravureRegiOn_HMI_i = FALSE THEN uiState_2:=0;	END_IF
	
	40:// THE REGISTER IS LOCKED
		
			//Enable PI controller
			bPauseRegiOn_HMI_i := FALSE;
				
			IF NOT arAxisStatus_gb[Drive1.AxisNo].SyncMode.PhasingSlaveDone THEN	uiState_2:=35;	END_IF
				
			IF 	bGravureRegiOn_HMI_i = FALSE THEN uiState_2:=0;	END_IF
END_CASE

END_PROGRAM

// IndraMotionMlc1/Application/AdjustPreset/AdjustPreset
PROGRAM AdjustPreset
VAR
	diPresetValue_i: DINT;
	fbJogInc: R_TRIG;
	fbJogDec: R_TRIG;
	fbRegAdv: R_TRIG;
	fbRegRet: R_TRIG;
	
	bAdjustingRetard :BOOL:=FALSE;
	bAdjustingAdvance :BOOL:=FALSE;
END_VAR

diPresetValue_i	:=	REAL_TO_DINT(rSetPointWindows_gb * 10000.0);

bGravure_Jog_Adv_HMI_i;
bGravure_Jog_Ret_HMI_i;
diPresetValue_i;

rSetPointWindows_gb; // the value found when opening window

fbJogInc(CLK:=bGravure_Jog_Adv_HMI_i , Q=>  );
IF fbJogInc.Q THEN rSetPointWindows_gb := rSetPointWindows_gb + (0.0218*5.0); END_IF	//5mils adjustments
fbJogDec(CLK:=bGravure_Jog_Ret_HMI_i , Q=> );
IF fbJogDec.Q THEN rSetPointWindows_gb := rSetPointWindows_gb - (0.0218*5.0); END_IF	//5mils adjustments


//PROBLEM INPUT_RANGE_ERROR found on 11july2014
IF ModbusCom.rStepWidth > 0.0 AND ModbusCom.rStepWidth < 10.0 AND arAxisStatus_gb[Drive1.AxisNo].Admin._OpModeAck = ModeSyncPhase THEN	
	arAxisCtrl_gb[Drive1.AxisNo].SyncMode.AdjPhaseOffset.StepWidth:=	ModbusCom.rStepDeg;
ELSE 
	arAxisCtrl_gb[Drive1.AxisNo].SyncMode.AdjPhaseOffset.StepWidth			:= 1.0;
END_IF


//IMPORTANT!!!
//CORRECTION ON GRAVURE MUST BE DONE WHEN GRAVURE NIP IS OFF
//fbRegAdv(CLK:=bRegAdvance_ETH_i AND NOT bGravureNipActive_i , Q=>  );
//IF fbRegAdv.Q AND NOT bAdjustingAdvance AND NOT bAdjustingRetard THEN 
//rSetPointWindows_gb := rSetPointWindows_gb + ModbusCom.rStepDeg;
//arAxisCtrl_gb[Drive1.AxisNo].SyncMode.AdjPhaseOffset.Inc :=  TRUE;
//bAdjustingAdvance := TRUE;
//ELSIF arAxisStatus_gb[Drive1.AxisNo].SyncMode.PhasingSlaveDone THEN
//arAxisCtrl_gb[Drive1.AxisNo].SyncMode.AdjPhaseOffset.Inc := FALSE; 
//bAdjustingAdvance := FALSE;
//END_IF	//5mils adjustments
//AFTER ADJUSTING PHASEOFFSET WE MUST ADJUST THE WINDOW


//IMPORTANT!!!
//CORRECTION ON GRAVURE MUST BE DONE WHEN GRAVURE NIP IS OFF
//fbRegAdv(CLK:=bRegAdvance_ETH_i AND NOT bGravureNipActive_i , Q=>  );
//fbRegRet(CLK:=bRegRetard_ETH_i  AND NOT bGravureNipActive_i , Q=> );
fbRegAdv(CLK:=bRegAdvance_ETH_i  , Q=>  );
fbRegRet(CLK:=bRegRetard_ETH_i   , Q=> );
IF fbRegAdv.Q AND NOT bAdjustingAdvance AND NOT bAdjustingRetard THEN 
rSetPointWindows_gb := rSetPointWindows_gb + ModbusCom.rStepDeg;
arAxisCtrl_gb[Drive1.AxisNo].SyncMode.AdjPhaseOffset.Inc :=  TRUE;
bAdjustingAdvance := TRUE;
ELSIF fbRegRet.Q AND NOT bAdjustingAdvance AND NOT bAdjustingRetard THEN
rSetPointWindows_gb := rSetPointWindows_gb - ModbusCom.rStepDeg;
arAxisCtrl_gb[Drive1.AxisNo].SyncMode.AdjPhaseOffset.Dec := TRUE;
bAdjustingRetard := TRUE;
ELSIF arAxisStatus_gb[Drive1.AxisNo].SyncMode.PhasingSlaveDone THEN

arAxisCtrl_gb[Drive1.AxisNo].SyncMode.AdjPhaseOffset.Inc := FALSE;
arAxisCtrl_gb[Drive1.AxisNo].SyncMode.AdjPhaseOffset.Dec := FALSE;
bAdjustingRetard := FALSE;
bAdjustingAdvance := FALSE; 
END_IF	//5mils adjustments
//AFTER ADJUSTING PHASEOFFSET WE MUST ADJUST THE WINDOW

END_PROGRAM

// IndraMotionMlc1/Application/MAIN_PGM/ModbusCom
PROGRAM ModbusCom
(* Run in a low priority task *)
VAR
	fb_IL_ModBusTCPServerType02: IL_ModBusTCPServerType02; (* Instance of function block IL_ModbusTCPServerType02       *)	
	// Enable function block IL_ModbusTCPServerType02
	bEnableModbusSrv: BOOL := true;
	wPortNumber:           WORD := 502;                (* Modbus server port - 502 is Modbus default                    *)
	arbyBitData:           ARRAY[0..50] OF BYTE;     (* Coil data area for FC2, FC5 and FC15                          *)
	arbyDiscreteInputs:    ARRAY[0..50] OF BYTE;     (* Discrete Input data area for FC1  (read only)                 *)
	RegisterData:          REGISTER_DATA;              (* Holding Register data area for FC3, FC6, FC16 and FC23        *)
	InputRegisters:        REGISTER_DATA;              (* Input Register data area for FC4  (read only)                 *)
	bInOperation:          BOOL;                       (* Function block IL_ModbusTCPServer is in operation             *)
	bError:                BOOL;                       (* Function block IL_ModbusTCPServer quits operation with error  *)
	ErrorID:               ERROR_CODE;                 (* general information about the error                           *)
	ErrorIdent:            ERROR_STRUCT;               (* detailed information about the error                          *)
	Stats:                 IL_MODBUS_STATS;            (* connection statistics                                         *)

	(* test variables *)
	pdwBitData_998:        POINTER TO DWORD;           (* pointer to modify some bytes of RegisterData                  *)
	udiCycleCount:         UDINT;                      (* internal PLC cycle counter                                    *)
	bInit:                 BOOL := TRUE;               (* indicator for first start of PLC                              *)
	i:                     INT;                        (* internal loop counter                                         *)
	pdwBitData_2: POINTER TO WORD;
	bInfeed_Inc_Tens_HMI: INT;
	rStepWidth:REAL:=1.0;
	rStepCorrection:REAL:=10.0; //10 millieme
	rStepDeg:REAL;
	j:INT;
	k:INT;
END_VAR

j:= j+1;

fb_IL_ModBusTCPServerType02(
	Enable := bEnableModbusSrv,
	Port := wPortNumber,
	CoilData:= ADR(arbyBitData), 
	SizeOfCoilData:= SIZEOF(arbyBitData), 
	InputData:= ADR(arbyDiscreteInputs), 
	SizeOfInputData:= SIZEOF(arbyDiscreteInputs), 
	HoldingRegisterData:= ADR(RegisterData),
	SizeOfHoldingRegisterData:= SIZEOF(RegisterData), 
	InputRegisterData:= ADR(InputRegisters), 
	SizeOfInputRegisterData:= SIZEOF(InputRegisters), 
	InOperation => bInOperation,
	Error => bError,
	ErrorID => ErrorID,
	ErrorIdent => ErrorIdent,
	Stats => Stats);
	


	k:= k+1;
	

//GRAVURE FROM M258
bRegAdvance_ETH_i							:= RegisterData.arWord[10].2;
bRegRetard_ETH_i							:= RegisterData.arWord[10].3;
bGravureOn_ETH_q 							:= RegisterData.arWord[10].4;
bGravure_ResetDrive_HMI_i 		:=	RegisterData.arWord[10].5;
bRewindPID_Out_i							:=	RegisterData.arWord[10].6;
bGravureSlowRot_ETH_i					:=	RegisterData.arWord[10].7;
bGravureRegiOn_HMI_i					:=	RegisterData.arWord[10].8;
bGravure_Jog_Adv_HMI_i					:=	RegisterData.arWord[10].9;
bGravure_Jog_Ret_HMI_i					:=	RegisterData.arWord[10].10;
bInfeedRegiOn_HMI_i						:=	RegisterData.arWord[10].11;
bGravureNipActive_i						:=	RegisterData.arWord[10].12;


//STATUS TO M258 PLC
//bGravure_StatusSynch_HMI_q		:= arAxisStatus_gb[Drive1.AxisNo].Admin._OpModeAck = ModeAB;
(*GRAVURE STATUS*)
IF arAxisStatus_gb[Drive1.AxisNo].Diag.Error = TRUE THEN
	bGravure_StatusDisabled_HMI_q 	:= FALSE;
	bGravure_StatusSlowRot_HMI_q 	:= FALSE;
	bGravure_StatusSynch_HMI_q		:= FALSE;
	bGravure_StatusError_HMI_q		:= TRUE;
ELSIF (arAxisStatus_gb[Drive1.AxisNo].Admin._OpModeAck) = MODEVEL THEN
	bGravure_StatusDisabled_HMI_q 	:= FALSE;
	bGravure_StatusSlowRot_HMI_q 	:= TRUE;
	bGravure_StatusSynch_HMI_q		:= FALSE;
	bGravure_StatusError_HMI_q		:= FALSE;
ELSIF (arAxisStatus_gb[Drive1.AxisNo].Admin._OpModeAck) = MODESYNCPHASE THEN
	bGravure_StatusDisabled_HMI_q 	:= FALSE;
	bGravure_StatusSlowRot_HMI_q 	:= FALSE;
	bGravure_StatusSynch_HMI_q		:= TRUE;
	bGravure_StatusError_HMI_q		:= FALSE;
ELSE
	bGravure_StatusDisabled_HMI_q 	:= FALSE;
	bGravure_StatusSlowRot_HMI_q 	:= FALSE;
	bGravure_StatusSynch_HMI_q		:= FALSE;
	bGravure_StatusError_HMI_q		:= FALSE;
END_IF
RegisterData.arWord[2].0	:= bGravure_StatusDisabled_HMI_q;
RegisterData.arWord[2].1	:= bGravure_StatusSlowRot_HMI_q	;
RegisterData.arWord[2].2	:= bGravure_StatusSynch_HMI_q	;
RegisterData.arWord[2].3	:= bGravure_StatusError_HMI_q;




 
//rDeviationMil_gb	:= ((rDeviation_gb*360.0)/16541.7)1000.0
rDeviationMil_gb		:= ((rDeviation_gb)*16541.7)/360.0/1000.0;
rSetPointWindowsMil_gb	:= ((rSetPointWindows_gb)*16541.7)/360.0/1000.0;

//DEVIATION
RegisterData.arWord[3]	:= DWORD_TO_WORD(dwDeviation_low_gb);
RegisterData.arWord[4]	:= DWORD_TO_WORD(SHR(dwDeviation_high_gb,16));

//CONTROL SETPOINT
RegisterData.arWord[5]	:= DWORD_TO_WORD(dwRegiCtrlSetPoint_low_gb);
RegisterData.arWord[6]	:= DWORD_TO_WORD(SHR(dwRegiCtrlSetPoint_high_gb,16));


//**************************************************************************
//**INFEED
//**************************************************************************
//INFEED FROM M258
bInfeed_Inc_Tens_HMI_i	:= RegisterData.arWord[12].0;
bInfeed_Dec_Tens_HMI_i	:= RegisterData.arWord[12].1;
bInfeedOn_ETH_q			:= RegisterData.arWord[12].2;
bInfeedManual_ETH_q		:= RegisterData.arWord[12].3;
bInfeed_ResetDrive_HMI_i :=  RegisterData.arWord[12].4;
//arAxisCtrl_gb[Drive2.AxisNo].Admin.ClearError	:=  bInfeed_ResetDrive_HMI_i 	OR x1;	//Reset HSC1.1 Infeed
//arAxisCtrl_gb[VMA_FT.AxisNo].Admin.ClearError	:=  bInfeed_ResetDrive_HMI_i	OR x1;	//Reset HSC1.1 Infeed
ImcCtrl.Admin.ClearError						:=  bGravure_ResetDrive_HMI_i OR bInfeed_ResetDrive_HMI_i 	OR x1;	//AxisInterface






dwRegAdjustLow_gb	:= WORD_TO_DWORD(RegisterData.arWord[13]);
dwRegAdjustHigh_gb	:= SHL(WORD_TO_DWORD(RegisterData.arWord[14]),16);
dwRegAdjust_gb		:= dwRegAdjustLow_gb OR dwRegAdjustHigh_gb;
rStepCorrection		:= DWORD_TO_REAL(dwRegAdjust_gb);

//THIS MAKE IT EDGED CONTROLLED
arAxisCtrl_gb[Drive1.AxisNo].SyncMode.AdjPhaseOffset.SelIncAdjust := TRUE;

//****** Hubert Crete_9th July 2014 ******
//FOR A GRAVURE OF 16541.7 mil
//1 mil = 0.0218 deg
//DIVISION BY 1000.0 is for readjustment since we multiplied by 1000.0 in the PLC_M258
(*	rStepDeg := ((rStepCorrection * 360.0)/16541.7)/1000.0;	



	arAxisCtrl_gb[Drive1.AxisNo].SyncMode.AdjPhaseOffset.Enable				:= TRUE;
(*	arAxisCtrl_gb[Drive1.AxisNo].SyncMode.AdjPhaseOffset.LowLimit			:=	0;
	arAxisCtrl_gb[Drive1.AxisNo].SyncMode.AdjPhaseOffset.HighLimit			:=	0;*)
	arAxisCtrl_gb[Drive1.AxisNo].SyncMode.AdjPhaseOffset.StepsPerSecond		:= 4;
	arAxisCtrl_gb[Drive1.AxisNo].SyncMode.AdjPhaseOffset.LowStepsPerSec		:= 10;
	arAxisCtrl_gb[Drive1.AxisNo].SyncMode.AdjPhaseOffset.LowStepWidth		:= 10;
	(*MUST SLOW DOWN GRAVURE ACCORDING TO DECIMAL VALUE HCP 9july2014*)
	arAxisCtrl_gb[Drive1.AxisNo].SyncMode.FineAdjust	:= -0.25;*)




//**************************************************************************
//INFEED FROM BOSCH MLC/L45 TO M258
//Load cell Tension
//RegisterData.arWord[7]	:= DWORD_TO_WORD(dwLoadcellTension_gb);
//RegisterData.arWord[8]	:= DWORD_TO_WORD(SHR(dwLoadcellTension_gb,16));



//RegisterData.arWord[0]	:= UINT_TO_WORD(InfeedState.uiInfeedGearing);
(*INFEED STATUS*)


IF arAxisStatus_gb[Drive2.AxisNo].Diag.Error = TRUE THEN
	bInfeed_StatusDisabled_HMI_q 	:= FALSE;
	bInfeed_StatusSlowRot_HMI_q 	:= FALSE;
	bInfeed_StatusSynch_HMI_q		:= FALSE;
	bInfeed_StatusError_HMI_q		:= TRUE;
ELSIF (arAxisStatus_gb[Drive2.AxisNo].Admin._OpModeAck) = ModeAB THEN
	bInfeed_StatusDisabled_HMI_q 	:= TRUE;
	bInfeed_StatusSlowRot_HMI_q 	:= FALSE;
	bInfeed_StatusSynch_HMI_q		:= FALSE;
	bInfeed_StatusError_HMI_q		:= FALSE;
ELSIF (arAxisStatus_gb[Drive2.AxisNo].Admin._OpModeAck) = MODEVEL THEN
	bInfeed_StatusDisabled_HMI_q 	:= FALSE;
	bInfeed_StatusSlowRot_HMI_q 	:= TRUE;
	bInfeed_StatusSynch_HMI_q		:= FALSE;
	bInfeed_StatusError_HMI_q		:= FALSE;
ELSIF (arAxisStatus_gb[Drive2.AxisNo].Admin._OpModeAck) = MODESYNCPHASE THEN
	bInfeed_StatusDisabled_HMI_q 	:= FALSE;
	bInfeed_StatusSlowRot_HMI_q 	:= FALSE;
	bInfeed_StatusSynch_HMI_q		:= TRUE;
	bInfeed_StatusError_HMI_q		:= FALSE;
ELSE
	bInfeed_StatusDisabled_HMI_q 	:= FALSE;
	bInfeed_StatusSlowRot_HMI_q 	:= FALSE;
	bInfeed_StatusSynch_HMI_q		:= FALSE;
	bInfeed_StatusError_HMI_q		:= FALSE;
END_IF
RegisterData.arWord[9].0	:= bInfeed_StatusDisabled_HMI_q;
RegisterData.arWord[9].1	:= bInfeed_StatusSlowRot_HMI_q	;
RegisterData.arWord[9].2	:= bInfeed_StatusSynch_HMI_q	;
RegisterData.arWord[9].3	:= bInfeed_StatusError_HMI_q;	
//ImcStatus.Diag.Error;						//vershmi
//arAxisStatus_gb[Drive1.AxisNo].Diag.Error;	//vershmi
arAxisCtrl_gb[Drive1.AxisNo].Admin.ClearError	:=	bGravure_ResetDrive_HMI_i OR x1;	//duhmiversmotion




x1;
x2;
x3;
x4;
x5;
x6;
x7;
x8;

END_PROGRAM

// IndraMotionMlc1/Application/AdjustPreset/WriteExpectWindow
PROGRAM WriteExpectWindow
VAR
	
	diDeadTimeCompensation: DINT;
			bPreset: BOOL;
	rPresetValue: REAL;
	rStepWidth:REAL:= 1.0;
	rStepSecond:REAL:= 1.0;
	
	arr1 : ARRAY [1..5] OF INT := [1,2,3,4,5];

	arTimeIntervals: ARRAY [1..4] OF REAL := [1.0,1.0,1.0,1.0];
	arWeightFactor: ARRAY [1..5] OF REAL := [1.0,1.0,1.0,1.0,1.0];
	arTimeInterAdjust: ARRAY [1..4] OF REAL := [1.0,1.0,1.0,1.0];(*Array of Time values for Cont Adjust FBs*)
	arWeightFacAdjust: ARRAY [1..5] OF REAL := [1.0,1.0,1.0,1.0,1.0];(*Array of Factor for Cont Adjust FBs*)
	
	
fbTouchProbeCont: MB_TouchProbeContinuous;
	bTouchProbeInOp: BOOL;
	bTouchProbeError: BOOL;
	fbRegiCtrl: MB_RegisterControllerType04;
	bPauseRegiCtrl: BOOL;
	bPresetRegiCtrl: BOOL;
	bDisableCyclicRegiCtrl: BOOL :=TRUE;
	bSetPtLckRegiCtrl: BOOL;
	BClearMemRegiCtrl: BOOL;
	bPolRegiCtrl: BOOL;
	rPGainRegiCtrl: REAL	:= 0.8;
	rIGainRegiCtrl: REAL	:= 10.0;
	rTCtrlRegiCtrl: REAL;
	rCorrStart: REAL;
	rCorrEnd: REAL := 270;
	arRespCurve: ARRAY [0..3] OF IL_COORD_TYPE01 := [3((X := 1, Y := 1)), (X := 0.0, Y := 0.0)];
	
	bRegiCtrlInOp: BOOL;
	bRegiCtrlError: BOOL;
	bRegiCtrlPaused: BOOL;
	bRegiCtrlPresetOK: BOOL;
	bHiLimActive: BOOL;
	bLowwLimActive: BOOL;
	rControlVal: REAL;
	rCurrentVal: REAL;
	rRegiCtrlDeviation: REAL;
	rParValRegiCtrl: REAL;
	fbtrigOpenWindows: R_TRIG;
	fbtrigCloseWindows: R_TRIG;
	uiMarkGating: UINT := 0;
	fbRegiCtrl02: MB_RegisterControllerType02;

	bset:BOOL;
	
	bPause:BOOL;
	bSetPtLock:BOOL;
//	bPauseRegiOn_HMI_i OR bSetPtLckRegiCtrl_HMI_i
	rSetPointWindows_gb2: REAL;
	
		rDeviationPos_gb:REAL;
	rDeviationBack_gb: REAL;
	
	rRegiCtrlSetPointPos_gb:REAL;
	fbContinuousAdjust: MB_ContinuousAdjustType01;
	bAutoContinuousAdj_ON: BOOL;
	
	
	rLatchedPosEdge: REAL;
	

	
	fbWriteExpectWindow: MB_WriteExpectWindow;
	fbRtrig_RegiCtrl: R_TRIG;
	fbContAdj: MB_ContinuousAdjustType02;

	diJogRefence:DINT;
	bAdjustRedCmd: BOOL;
	bEnableRegister:BOOL;
	fbFtrig: F_TRIG;
	
	diRealValue:DINT;
	rRealValue:REAL;
	rRealValue1:REAL;
	rRealValue2:REAL;
	diCurrentValue:DINT;
	diPresetValue_i: DINT;
	
	rVar: REAL;
	bSetPtLckRegiCtrl_HMI_i2: BOOL;
END_VAR

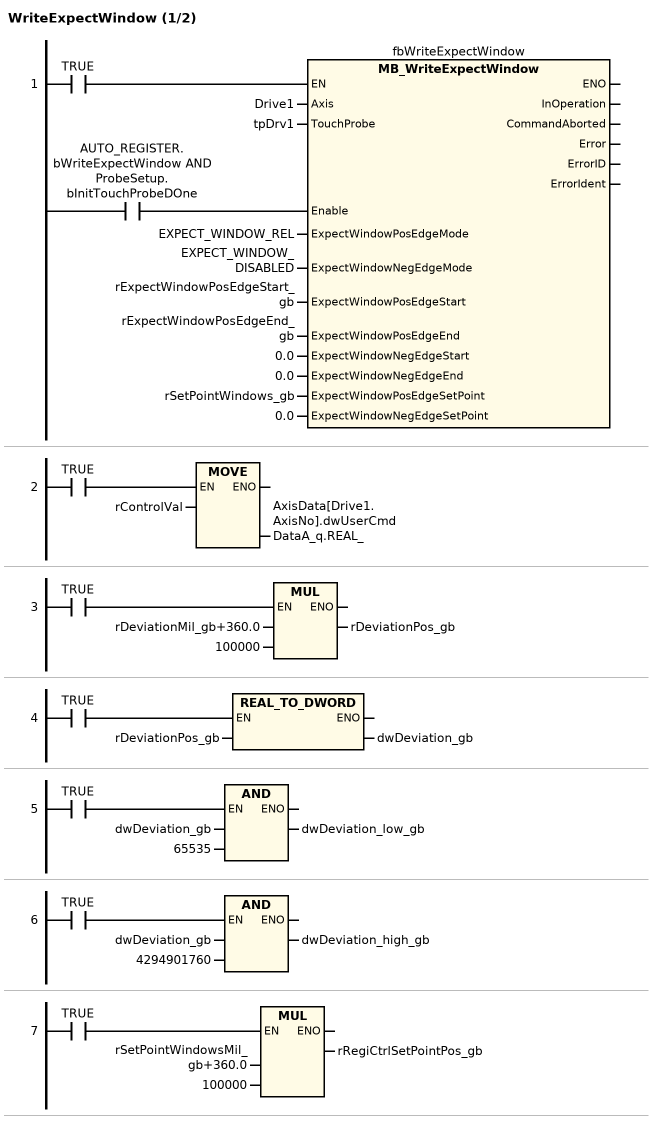
// NETWORK 1
//   Drive1: Real axis "Drive1" with axis number 1
//   tpDrv1: FALSE: PlcProg is active DEFINITION DU TOUCHPROB
//   EXPECT_WINDOW_DISABLED: expectation window disabled
fbWriteExpectWindow(
    Axis := Drive1,
    TouchProbe := tpDrv1,
    Enable := AUTO_REGISTER.bWriteExpectWindow AND ProbeSetup.bInitTouchProbeDOne,
    ExpectWindowPosEdgeMode := EXPECT_WINDOW_REL,
    ExpectWindowNegEdgeMode := EXPECT_WINDOW_DISABLED,
    ExpectWindowPosEdgeStart := rExpectWindowPosEdgeStart_gb,
    ExpectWindowPosEdgeEnd := rExpectWindowPosEdgeEnd_gb,
    ExpectWindowNegEdgeStart := 0.0,
    ExpectWindowNegEdgeEnd := 0.0,
    ExpectWindowPosEdgeSetPoint := rSetPointWindows_gb,
    ExpectWindowNegEdgeSetPoint := 0.0); // MB_WriteExpectWindow

// NETWORK 2
AxisData[Drive1.AxisNo].dwUserCmdDataA_q.REAL_ := rControlVal;

// NETWORK 3
rDeviationPos_gb := (rDeviationMil_gb+360.0) * 100000;

// NETWORK 4
dwDeviation_gb := REAL_TO_DWORD(rDeviationPos_gb);

// NETWORK 5
dwDeviation_low_gb := dwDeviation_gb AND 65535;

// NETWORK 6
dwDeviation_high_gb := dwDeviation_gb AND 4294901760;

// NETWORK 7
rRegiCtrlSetPointPos_gb := (rSetPointWindowsMil_gb+360.0) * 100000;

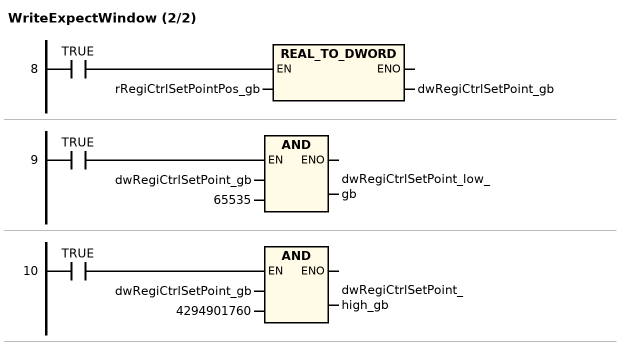
// NETWORK 8
dwRegiCtrlSetPoint_gb := REAL_TO_DWORD(rRegiCtrlSetPointPos_gb);

// NETWORK 9
dwRegiCtrlSetPoint_low_gb := dwRegiCtrlSetPoint_gb AND 65535;

// NETWORK 10
dwRegiCtrlSetPoint_high_gb := dwRegiCtrlSetPoint_gb AND 4294901760;

END_PROGRAM

// IndraMotionMlc1/Application/FLEXO_PGM/ProbeSetup
PROGRAM ProbeSetup
VAR
	
	
	//new: ARRAY[0..20] OF MB_InitTouchProbe;
	//new:	MB_InitTouchProbe;
	FB: ARRAY[1..20] OF MB_InitTouchProbe;
	bInitTouchProbe: ARRAY[1..20] OF BOOL;
	ExpectWindowPosEdgeSetPoint: INT;
	ExpectWindowNegEdgeSetPoint: INT;
	MarkerFailureEnable: BOOL;
	MaxNumberOfMarkerFailure: INT;
	Interpolation: INT;
	TimeStampEnable: BOOL;
	DeadTimePosEdge: INT;
	DeadTimeNegEdge: INT;
	ProbeData: INT;
	PositionEvalMode: INT;
	Axis: AXIS_REF;
	TouchProbe: TOUCHPROBE_REF;
	Done: BOOL;
	
	commanddone:BOOL;
	index :UINT;
	bInitTouchProbeDOne:BOOL;
	
END_VAR

VAR_INPUT
	
END_VAR


//FOR index:=1 TO uiPRINT_AXIS_INDEX BY 1 DO
FOR index:=1 TO 2 BY 1 DO

FB[index](
	Execute:= ImcStatus.Admin.ModeStatus_BB, 
	ProbeModule:= , 
	ExecutionMode:= MB_EXECUTION_MODE.EXECUTE_CYCLIC , 
	ProbeInput:= , 
	ExpectWindowPosEdgeMode:= EXPECT_WINDOW_REL ,
	ExpectWindowNegEdgeMode:= EXPECT_WINDOW_DISABLED, 
	ExpectWindowPosEdgeStart:= 179.999, 
	ExpectWindowPosEdgeEnd:= 179.999, 
	ExpectWindowNegEdgeStart:= 0, 
	ExpectWindowNegEdgeEnd:= 0, 
	ExpectWindowPosEdgeSetPoint:= 180, 
	ExpectWindowNegEdgeSetPoint:= 0, 
	MarkerFailureEnable:= FALSE, 
	MaxNumberOfMarkerFailure:= 0, 
	Interpolation:= MB_INTERPOLATION_MODE.NO_INTERPOLATION, 
	TimeStampEnable:= FALSE, 
	DeadTimePosEdge:= 30, 
	DeadTimeNegEdge:= 0, 
	ProbeData:=MB_PROBE_DATA.TP_ACT_POS_FEEDBACK1 , 
	PositionEvalMode:=MB_POSITION_EVAL.POSITION_POS_EDGE , 
	DiffEvalMode:= MB_DIFF_EVAL.DIFF_DISABLED, 
	Axis:= arDrive[1], 
	TouchProbe:= arProbe[index], 
	Done=> bInitTouchProbe[index], 
	Active=> , 
	Error=> , 
	ErrorID=> , 
	ErrorIdent=> );
END_FOR;

END_PROGRAM

// IndraMotionMlc1/Application/FLEXO_PGM/TouchProbe
PROGRAM TouchProbe
VAR
	PaperPos: MB_TouchProbeContinuous;
	MarkPos:	MB_TouchProbeContinuous;
	
	bReadyToExec: BOOL;
	bGoProbe:BOOL;
	rLatchPos:REAL;
	
	fbPaperWindow: MB_WriteExpectWindow;
	bExecWindow: BOOL;
	
	rSetpoint:REAL;
	rPaperStartWin:REAL;
	rPaperStopWin:REAL;
	rMarkStartWin:REAL;
	rMarkStopWin:REAL;
	
	rEffectiveStartWin:REAL;
	rEffectiveStopWin:REAL;
	rCheckStart:REAL;
	
	//fbWindowExec: TP;
	fbWindowExec: TON;
	
	bPaperExec:BOOL;
	bMarkExec:BOOL;
	rStartWin: LREAL;
	rPrintOffsetPos : REAL := 120.0;
	rLatchPos1: REAL;
	rLatchPos2: REAL;
	rDeltaPos:REAL;
	rPaperPos: REAL;
	rMarkPos: REAL;

	FB_WritePaperStartWin: MB_WriteRealParameter;
	FB_WritePaperStopWin: MB_WriteRealParameter;
	FB_WriteMarkStartWin: MB_WriteRealParameter;
	FB_WriteMarkStopWin: MB_WriteRealParameter;
	
	bToggle:BOOL;
	bInitCom:BOOL;
	bWriteThat:BOOL;
	rRamdomThat:REAL := 0.01;
	WritePar: TP ;
	
	
	
	writevar1: FB_writevar;
	writevar2: FB_writevar;
	writevar3: FB_writevar;
	writevar4: FB_writevar;
END_VAR



//bReadyToExec:=ProbeSetup.bInitTouchProbeDOne AND ImcStatus.Admin.ModeStatus_BB AND bGoProbe;

bPaperExec := ProbeSetup.bInitTouchProbe[1] AND ImcStatus.Admin.ModeStatus_BB AND bGoProbe;
bMarkExec := ProbeSetup.bInitTouchProbe[2] AND ImcStatus.Admin.ModeStatus_BB AND bGoProbe;

PaperPos(
	Enable:=bPaperExec , 
	Axis:=  arDrive[1], 
	TouchProbe:= arProbe[1], 
	InOperation=> , 
	CommandAborted=> , 
	Error=> , 
	ErrorID=> , 
	ErrorIdent=> , 
	DetectedPosEdge=> , 
	DetectedNegEdge=> , 
	RecordedPositionPosEdge=>  rPaperPos, 
	RecordedPositionNegEdge=> , 
	PositionDifference=> , 
	DetectedPositionDifference=> , 
	MissingMarksPosEdge=> , 
	MissingMarksNegEdge=> , 
	TimeStampPosEdge=> , 
	TimeStampNegEdge=> );
	
MarkPos(
	Enable:=bMarkExec , 
	Axis:=  arDrive[1], 
	TouchProbe:= arProbe[2], 
	InOperation=> , 
	CommandAborted=> , 
	Error=> , 
	ErrorID=> , 
	ErrorIdent=> , 
	DetectedPosEdge=> , 
	DetectedNegEdge=> , 
	RecordedPositionPosEdge=>  rMarkPos, 
	RecordedPositionNegEdge=> , 
	PositionDifference=> , 
	DetectedPositionDifference=> , 
	MissingMarksPosEdge=> , 
	MissingMarksNegEdge=> , 
	TimeStampPosEdge=> , 
	TimeStampNegEdge=> );	
	

	
	
	
	IF PaperPos.DetectedPosEdge >= 1 AND PaperPos.InOperation THEN
		rPaperStartWin := 	rPaperPos -5.0;
		rPaperStopWin := 	rPaperPos +5.0;
		
		IF rPaperPos > 180.0 THEN 
			rMarkStartWin	:= (rPaperPos -5.0 -rPrintOffsetPos);
			rMarkStopWin	:= (rPaperPos +5.0 -rPrintOffsetPos);
		ELSE
			rMarkStartWin	:= (rPaperPos -5.0 +rPrintOffsetPos);
			rMarkStopWin	:= (rPaperPos +5.0 +rPrintOffsetPos);
		END_IF
	ELSE
		rPaperStartWin 	:= 0.01;
		rPaperStopWin	:=	359.9;
		rMarkStartWin 	:= 179.9;
		rMarkStopWin	:=	180.0;
		
	END_IF
	
	

	writevar1(bStartWriting:=bWriteThat , rValueToWrite:= rPaperStartWin, stParameter:=GVL_P_Param_ID.FP_P_0_0204 );
	writevar2(bStartWriting:=bWriteThat , rValueToWrite:= rPaperStopWin, stParameter:=GVL_P_Param_ID.FP_P_0_0205 );
	writevar3(bStartWriting:=bWriteThat , rValueToWrite:= rMarkStartWin, stParameter:=GVL_P_Param_ID.FP_P_0_0200 );
	writevar4(bStartWriting:=bWriteThat , rValueToWrite:= rMarkStopWin, stParameter:=GVL_P_Param_ID.FP_P_0_0201 );
	
	IF MarkPos.InOperation AND PaperPos.InOperation AND rMarkPos <> 0.0 AND rPaperPos<>0.0 THEN	
		IF rPaperPos < rMarkPos THEN 
			rDeltaPos := rPaperPos-rMarkPos + (rPrintOffsetPos*2.0);
		ELSE
			rDeltaPos := rPaperPos-rMarkPos;
		END_IF
	END_IF

END_PROGRAM

// IndraMotionMlc1/Application/Utilities/FB_writevar
FUNCTION_BLOCK FB_writevar
VAR
	uiState: INT;
	FB_WriteRealPar: MB_WriteRealParameter;
	bWriteExec:BOOL;
END_VAR

VAR_INPUT
	bStartWriting:BOOL;
	rValueToWrite:REAL;
	stParameter:MB_IDN;
END_VAR


CASE uiState OF
	
	0:
		bWriteExec := FALSE;
		IF bStartWriting = TRUE THEN
			uiState:= 1;
		END_IF
		
	1:
		bWriteExec := TRUE;
		IF (FB_WriteRealPar.Done) THEN
			uiState:= 2;
		END_IF
		
	
	2:
		bWriteExec:= FALSE;
		IF NOT FB_WriteRealPar.Done AND NOT FB_WriteRealPar.Active THEN
			uiState:= 0;
		END_IF
END_CASE

FB_WriteRealPar(
	Execute:=bWriteExec , 
	ParameterNumber:=stParameter , 
	Value:= rValueToWrite, 
	Axis:=  arDrive[1], 
	Done=> , 
	Active=> , 
	Error=> , 
	ErrorID=> , 
	ErrorIdent=> );

END_FUNCTION_BLOCK

// IndraMotionMlc1/Application/InsetterControl
PROGRAM InsetterControl
VAR
	fbRegiCtrlType02: MB_RegisterControllerType02
;
	bPreset: BOOL;
	fbTpCont: MB_TouchProbeContinuous;
	fbTouchProbeCont:MB_TouchProbeContinuous;
	bRegiCtrlOn: BOOL;
	bDisCyclic: BOOL;
	bSetPtLck: BOOL;
	bClrMeas: BOOL;
	bCtrlPol: BOOL;
	rPCtrl: REAL;
	rICtrl: REAL;
	rTCtrl: REAL;
	
	rRegisterCommand: REAL;
	arRespCurve: ARRAY [0..3] OF IL_COORD_TYPE01 := [4((X := 1, Y := 1))];
	
	rPresetValue: REAL;
	fbTpOneShot: MB_TouchProbe;
	bSingleShotProbe: BOOL;
	new:BOOL;
	fbProbeCnt: CTU;
	fbTrigCntProbe: R_TRIG;
	bRegiCtrlPause: BOOL;
	fbRegiMeasuring1: MB_RegiMeasuringType01;
	fbRegiRegulate1: MB_RegiRegulateType01;
	bEnableRegul1: BOOL;
	bPresetRegul1: BOOL;
	fbPITType02: IL_PIType02;
	rPCtrlPITType02: REAL := 2.0;
	rICtrlPITType02: REAL :=0.0;
	bProbeCont: BOOL;
	fbRegiRegulate2: MB_RegiRegulateType02;
	fbRegiRegulate3: MB_RegiRegulateType03;
	rWeighing: REAL := 1.0;
	bTpContFirstShot: BOOL;
	bTpOneShotSet: BOOL;
	uiLastProbeDectect: UINT;
	bProbeDetected: BOOL;
	fbCProbePos: R_TRIG;
	fbCProbePosFirst: R_TRIG;
	bStep_Triggered: BOOL;
	fbCntChk: CTU;
	fbTrigStep: R_TRIG;
	rLastRegulateRatio: REAL;
	bTransferUnLock: BOOL;
	rFineGearRatioAdjust: REAL;
	uiLastStepRegiDetected: INT;
	bRegiStepDetected: BOOL;
	fbRegiStepDetect: R_TRIG;
	bRegiStepTriggered: BOOL;
	bEnableIntegrator: BOOL;
	//fbIntegrator: FB_REGULATE_INTEGRATOR;
	lrMasterPosDeg: LREAL;
	bDisableCyclicP694: BOOL;
	bPresetIntegrator: BOOL;
	bPresetP694: BOOL;
		fbSetPointLck: MB_RegiSetpointLockType01;
	bSetPointLck: BOOL;
	rSetpoint: REAL;
	rDeviationPct: REAL;
	rDeviationRegiMeasuring_gb:REAL;
	uiProbeCnt: INT;
	arOfRecorderPos: ARRAY[0..101] OF real;
	rExpWinStart: REAL;
	rExpWinEnd: REAL;
	fbT: TON;
	fbSetPointLckTimer: BOOL;
	fbRegiRegulate11: MB_RegiRegulateType01;
END_VAR

VAR_OUTPUT
	
END_VAR

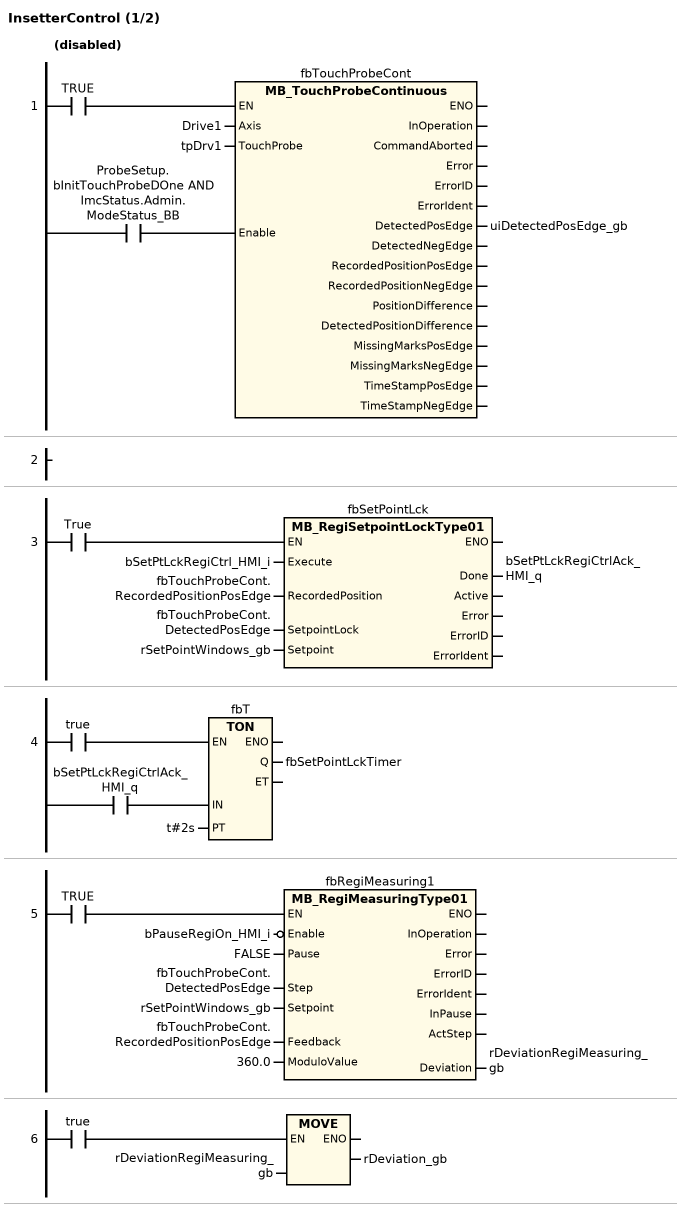
// NETWORK 1 (disabled)
//   Drive1: Real axis "Drive1" with axis number 1
//   tpDrv1: FALSE: PlcProg is active DEFINITION DU TOUCHPROB
// fbTouchProbeCont(
//     Axis := Drive1,
//     TouchProbe := tpDrv1,
//     Enable := ProbeSetup.bInitTouchProbeDOne AND ImcStatus.Admin.ModeStatus_BB,
//     DetectedPosEdge => uiDetectedPosEdge_gb); // MB_TouchProbeContinuous

// NETWORK 2

// NETWORK 3
//   fbTouchProbeCont.RecordedPositionPosEdge: Axis position where positive edge occurred (in degree)
//   fbTouchProbeCont.DetectedPosEdge: Positive edge of the selected probe was detected (reset if enable = FALSE)
IF True THEN
    fbSetPointLck(
        Execute := bSetPtLckRegiCtrl_HMI_i,
        RecordedPosition := fbTouchProbeCont.RecordedPositionPosEdge,
        SetpointLock := fbTouchProbeCont.DetectedPosEdge,
        Setpoint := rSetPointWindows_gb,
        Done => bSetPtLckRegiCtrlAck_HMI_q); // MB_RegiSetpointLockType01
END_IF

// NETWORK 4
IF true THEN
    fbT(IN := bSetPtLckRegiCtrlAck_HMI_q, PT := t#2s, Q => fbSetPointLckTimer); // TON
END_IF

// NETWORK 5
//   fbTouchProbeCont.DetectedPosEdge: Positive edge of the selected probe was detected (reset if enable = FALSE)
//   fbTouchProbeCont.RecordedPositionPosEdge: Axis position where positive edge occurred (in degree)
fbRegiMeasuring1(
    Enable := NOT bPauseRegiOn_HMI_i,
    Pause := FALSE,
    Step := fbTouchProbeCont.DetectedPosEdge,
    Setpoint := rSetPointWindows_gb,
    Feedback := fbTouchProbeCont.RecordedPositionPosEdge,
    ModuloValue := 360.0,
    Deviation => rDeviationRegiMeasuring_gb); // MB_RegiMeasuringType01

// NETWORK 6
IF true THEN rDeviation_gb := rDeviationRegiMeasuring_gb; END_IF

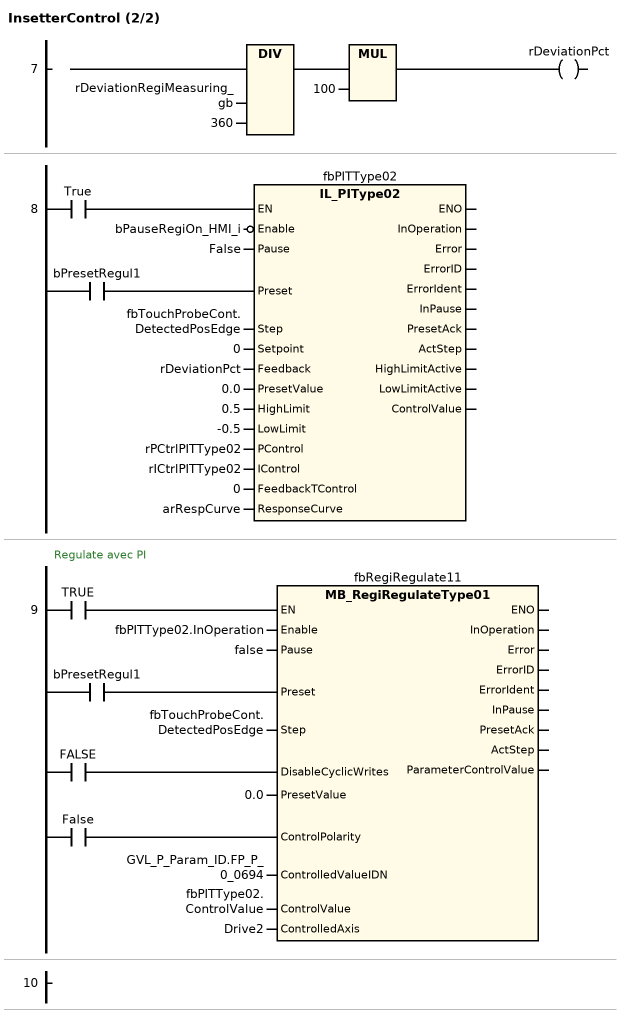
// NETWORK 7
rDeviationPct := (rDeviationRegiMeasuring_gb / 360) * 100;

// NETWORK 8
//   fbTouchProbeCont.DetectedPosEdge: Positive edge of the selected probe was detected (reset if enable = FALSE)
IF True THEN
    fbPITType02(
        Enable := NOT bPauseRegiOn_HMI_i,
        Pause := False,
        Preset := bPresetRegul1,
        Step := fbTouchProbeCont.DetectedPosEdge,
        Setpoint := 0,
        Feedback := rDeviationPct,
        PresetValue := 0.0,
        HighLimit := 0.5,
        LowLimit := -0.5,
        PControl := rPCtrlPITType02,
        IControl := rICtrlPITType02,
        FeedbackTControl := 0,
        ResponseCurve := arRespCurve); // IL_PIType02
END_IF

// NETWORK 9
// Regulate avec PI
//   fbPITType02.InOperation: If TRUE, the controller is working and the output is
//   fbTouchProbeCont.DetectedPosEdge: Positive edge of the selected probe was detected (reset if enable = FALSE)
//   fbPITType02.ControlValue: Calculated controller output value
//   Drive2: Real axis "Drive2" with axis number 3
fbRegiRegulate11(
    Enable := fbPITType02.InOperation,
    Pause := false,
    Preset := bPresetRegul1,
    Step := fbTouchProbeCont.DetectedPosEdge,
    DisableCyclicWrites := FALSE,
    PresetValue := 0.0,
    ControlPolarity := False,
    ControlledValueIDN := GVL_P_Param_ID.FP_P_0_0694,
    ControlValue := fbPITType02.ControlValue,
    ControlledAxis := Drive2); // MB_RegiRegulateType01

// NETWORK 10

END_PROGRAM

// IndraMotionMlc1/Application/POU
PROGRAM POU
VAR
	bBogus:BOOL;
	ii:UINT;
END_VAR

bBogus;
ii := ii+1;

IF TE_AxisInterfaceType01Prog.InitDone=FALSE THEN
	RETURN;
END_IF

//AXIS DEFINITION
arFlexoAxis[1] := arAxisCtrl_gb[Drive1.AxisNo].Admin.Axis;
arFlexoAxis[2] := arAxisCtrl_gb[Drive2.AxisNo].Admin.Axis;
//Winders
arWindingAxis[1]:= arAxisCtrl_gb[Drive20.AxisNo].Admin.Axis;

IF NOT binit THEN InitAxis(arAxisPointer:=ADR(arFlexoAxis) , uiNUM_FLEXO_F:= uiNUM_FLEXO);
				  InitAxis(arAxisPointer:=ADR(arWindingAxis) , uiNUM_FLEXO_F:= uiNUM_WINDER);

//ELSE	//______    INIT IS OVER       ______!!!!!!!



bReset_HMI_i;
//THIS FUNCTION IS THE CORE OF THE MACHINE POSSIBLE STATES
Winder(
	arAxisPointer:= ADR(arWindingAxis), 
	uiNUM_FLEXO_F:= uiNUM_WINDER, 
	MACHINE_STATE_i:= newSTATE, 
	iGearValue:= 1, 
	bRewIntrlock=> bRewIntrlock);


Machine(
	arAxisPointer_M	:=ADR(arFlexoAxis),
	uiNUM_FLEXO_M	:=uiNUM_FLEXO,
	bRun_i			:=	bRun_HMI_i , 
	bJog_i			:=	bJog_HMI_i , 
	bStop_i			:=	bStop_HMI_i , 
	okToRun			:=	bOkToRun_i , 
	okToJog			:=	bOkToJog_i , 
	bFault			:=	bFault_i, 
	bIntrlock		:=	bInterlock_i, 
	bSetup_i		:=	 bSetup_HMI_i,
	bWriteExec		:=  bWriteExec, 
	CURRENT_STATE_OUT=> newSTATE );	

rRepeat_i:=INT_TO_REAL(iFormat_i/iTeethConstant)/ 100.0;

//THIS FUNCTION SETS SPEED ACCORDING TO THE FORMAT 
SetVmaSpeed(
	arAxisPointer:=ADR(arFlexoAxis) , 
	uiNUM_FLEXO_F:=uiNUM_FLEXO , 
	rFormat:=rRepeat_i , 
	rRunSpeedDemandFPM:=rRunSpd , 
	rJogSpeedDemandFPM:= rJogSpd, 
	uiState:=newSTATE , 
	);
//SET FORMAT
//THIS FUNCTION SETS MECHANICAL GEAR DEPENDING ON THE PLATE CYLINDER USED
//IT ALSO ADJUSTS THE SYNC_REVOLUTION TO COMPENSATES THE ADJUSTMENT OF VMA SPEED
FormatC(
	arAxisPointer:= ADR(arFlexoAxis), 
	uiNUM_FLEXO_F:= uiNUM_FLEXO , 
	MACHINE_STATE_i:= newSTATE , 
	iGearValue:=     iFormat_i , 
	bExecute:= bWriteExec , 
	bSetupDone_i=> );

END_PROGRAM

// IndraMotionMlc1/Application/MOTION
PROGRAM MOTION
VAR
	arFlexoAxis:	ARRAY[1..20] OF AXIS_REF;
	arPullrollAxis: ARRAY[1..20] OF AXIS_REF;
	arWindingAxis:	ARRAY[1..20] OF AXIS_REF;
END_VAR


VAR CONSTANT
	uiNUM_FLEXO		: UINT	:= 2;
	uiNUM_PULLROLL	: UINT	:= 0;
END_VAR

TE_AxisInterfaceType01Prog();
MB_ImcInterface();

IF TE_AxisInterfaceType01Prog.InitDone=FALSE THEN
	RETURN;
END_IF


MAIN.rRepeat_i;

ProbeSetup(); //HCP_3107
TouchProbe();  //HCP_3107

WinderProcess(bWinder1Direction:=FALSE , bWinder2Direction:=FALSE , rRepeat_i:=MAIN.rRepeat_i );
//InsetterControl();

END_PROGRAM

// IndraMotionMlc1/Application/REWIND/WinderProcess
PROGRAM WinderProcess


VAR
	//bBogus: BOOL := FALSE;
	//bogus: BOOL;
	rTensionSetpointW1_HMI_i:REAL:= 10.0;
	
	bEnableWinder:BOOL;
    fbWindTension_W1: MB_WinderTensionCtrlType02;       (* winder with tension control for Winder #1 *)
	(*fbWindTension_W2: MB_WinderTensionCtrlType02;		(* winder with tension control for Winder #2*)*)
    fbDiameterMeasurement: MB_DiameterMeasurementType01;(* diameter measurement *)
    stWindTensDiagW1: MB_WIND_TENS_DIAG;                (* structure for wind tension diagnostics Winder #1 *)
	(*stWindTensDiagW2: MB_WIND_TENS_DIAG;                (* structure for wind tension diagnostics Winder #2 *)*)
    stWindTensDiamW1: MB_WIND_DIAMETER;					(* structure for wind tension diameter Winder #1 *)
	(*stWindTensDiamW2: MB_WIND_DIAMETER;					(* structure for wind tension diameter Winder #2 *)*)
	stWindTensionCtrlW1: MB_WIND_TENSION;
	(*stWindTensionCtrlW2: MB_WIND_TENSION;*)

    stWindFrictionW1: MB_WIND_FRICTION;         		(* structure for wind tension friction Winder #1 *)
	(*stWindFrictionW2: MB_WIND_FRICTION;         		(* structure for wind tension friction Winder #2 *)*)

	LowTimeTickWindTens: UDINT;                         (* winder tension measurement *)
	HighTimeTickWindTens: UDINT;                        (* winder tension time measurement *)
	TimeDiffWindTens: UDINT;                            (* winder tension time measurement *)
	TimeMaxWindTens: UDINT;                             (* winder tension time measurement *)

	(*Init Values *)
	rSetPointOpModeW1:REAL;								(* ANALOG1 SETPOINT *)
	rSetPointOpModeW2:REAL;								(* ANALOG2 SETPOINT *)
	rSetPointStandstillW1:REAL:=5.0;
	rSetPointStandstillW2:REAL:=5.0;
	rTensionSpeedW1: 	REAL := 10.0;
	rTensionSpeedW2:	REAL:=	10.0;
	rDefTorqueLimW1:REAL:=20.0;
	rDefTorqueLimW2:REAL:=20.0;
	rTensionInWindowW1:REAL:=20.0;
	rTensionInWindowW2:REAL:=20.0;
	tActualTorqFilterW1: TIME := T#50ms;		(* Filter time constant for the actual torque S-0-0084 "Torque/force feedback value"*)
	tActualTorqFilterW2: TIME := T#50ms;		(* Filter time constant for the actual torque S-0-0084 "Torque/force feedback value"*)
	tAccelTorqFilterW1: TIME :=  T#80ms;		(* Filter time constant for the acceleration torque*)
	tAccelTorqFilterW2: TIME :=  T#80ms;		(* Filter time constant for the acceleration torque*)
	rWindowInTensionPctW1: REAL := 30.0;		(* Window for the actual tension value [%] in relation to the command tension value*)
	rWindowInTensionPctW2: REAL := 30.0;		(* Window for the actual tension value [%] in relation to the command tension value*)
	rMinTensionMonitorW1: REAL := 5.0;			(* Lower threshold for the actual tension value (only for a display with binary output "MinTensionAck")*)
	rMinTensionMonitorW2: REAL := 5.0;			(* Lower threshold for the actual tension value (only for a display with binary output "MinTensionAck")*)
	rMaxTensionMonitorW1 : REAL := 100.0;		(* Upper threshold FOR the actual tension value (only FOR a display with binary output "MAX TensionAck"*)
	rMaxTensionMonitorW2 : REAL := 100.0;		(* Upper threshold FOR the actual tension value (only FOR a display with binary output "MAX TensionAck"*)
	
	//PRESENT ON SCREEN
	rStartDiameterW1_HMI: 				REAL 	:= 3.5;		//3.5 inchs.core
	rWinder1_Standstill_TensionHMI_gb:	REAL	:= 10.0;
	bNewRoll_Winder1_HMI_i:BOOL;

	(* array for Winder Recipes NOT INCLUDED IN FIRST VERSION SEPT2009*)
	//arWinderRecipes: ARRAY [0..31] OF WINDER_RECIPES;



	(*OUTPUTS FOR WINDER FUNCTION BLOCKS*)

	bPauseW1:					BOOL:= FALSE;
	bPauseW2:					BOOL:= FALSE;
	bInOperationW1: 			BOOL;
	bInOperationW2: 			BOOL;
	bErrorW1:					BOOL;
	bErrorW2:					BOOL;
	stErrorIdentW1:			ERROR_STRUCT;
	stErrorIdentW2:			ERROR_STRUCT;
	bInPauseW1:				BOOL;
	bInPauseW2:				BOOL;
	bPresetDiamAckW1:			BOOL;
	bPresetDiamAckW2:			BOOL;
	bInPauseDiamW1:			BOOL;
	bInPauseDiamW2:			BOOL;
	bMinAvDiamAchievedW1:		BOOL;
	bMinAvDiamAchievedW2:		BOOL;
	bMaxAvDiamAchievedW1:		BOOL;
	bMaxAvDiamAchievedW2:		BOOL;
	bHighLimitDiamActiveW1:	BOOL;
	bHighLimitDiamActiveW2:	BOOL;
	bLowLimitDiamActiveW1:	BOOL;
	bLowLimitDiamActiveW2:	BOOL;
	bDiameterEngagedW1:		BOOL;
	bDiameterEngagedW2:		BOOL;
	bHighLimitTensActiveW1:	BOOL;
	bHighLimitTensActiveW2:	BOOL;
	bLowLimitTensActiveW1:	BOOL;
	bLowLimitTensActiveW2:	BOOL;
	bTensionInWindowW1:		BOOL;
	bTensionInWindowW2:		BOOL;
	bMinTensionAchievedW1:	BOOL;
	bMinTensionAchievedW2:	BOOL;
	bMaxTensionAchievedW1:	BOOL;
	bMaxTensionAchievedW2:	BOOL;
	bDiameterBeginW1:		BOOL;
	bDiameterBeginW2:		BOOL;
	bDiameterFlagW1:		BOOL;
	bDiameterFlagW2:		BOOL;
	bFirstPresetW1:			BOOL:= TRUE;
	bFirstPresetW2:			BOOL;

	rCurrentDiameterW1: 		REAL;
	rCurrentDiameterW2: 		REAL;
	rGearRatioFineAdjustW1: 	REAL;
	rGearRatioFineAdjustW2: 	REAL;
	rCurrentInertiaW1: 			REAL;
	rCurrentInertiaW2: 			REAL;
	rSpeedOffsetW1: 			REAL;
	rSpeedOffsetW2: 			REAL;
	rTorqueLimitBipolarW1: 		REAL;
	rTorqueLimitBipolarW2: 		REAL;
	rActualTorqueW1: REAL;
	rActualTorqueW2: REAL;


	iDiameterAvg: UINT := 5;
	rWinderWebWidthRew1: REAL;
	rWinderWebWidthRew2: REAL;
	FTrig_DiameterEngaged: F_TRIG;

	(*PROCESS POTENTIOMETER VALUE *)

	rSetpointMaxW1				: REAL	:= 100.0;
	rSetpointProcessedW1		: REAL	:= 5.0;
	rCurrentDiameterProcessedW1	: REAL	:=	80.0;
	rSetpointMaxW2				: REAL	:= 100.0;
	rSetpointProcessedW2		: REAL	:= 5.0;
	rCurrentDiameterProcessedW2	: REAL	:=	80.0;

	rGearRatioFineAdjustW1_HMI:REAL;
	rSpeedOffsetW1_HMI:REAL;
	rCurrentDiameterW1_HMI:REAL;
	
	iVmAxisIdx: INT;

	rDensity: REAL;			(*Density Choosen *)
	wWebWidthRew1: WORD; 	(* Word for Binary width decoding *)
	wWebWidthRew2: WORD;
	rWebWidthRew1: REAL;
	rWebWidthRew2: REAL;
	rWebWidthInch1: REAL;
	rWebWidthInch2: REAL;

	fbCoreSizeRTRIG: R_TRIG;
	bMakeCoreSizeChange: BOOL := TRUE ;
	fbCoreSizeFTRIG: F_TRIG;
	
	rtemp: REAL;
	bOverloadW1: BOOL;
	bOverloadW2: BOOL;
	bWinder1_On_i_c: BOOL;
	bWinder2_On_i_c: BOOL;
	bWinder1_Dir_i_c: BOOL;
	bWinder2_Dir_i_c: BOOL;
	rWebWidthInch2Check: REAL;
	rWebWidthInch1Check: REAL;
	//fbEndOfRoll: FREQ_MEASURE;
	//fbUnwindFreq: FREQ_MEASURE;
	//fbInfeedFreq: FREQ_MEASURE;
	fbEndOfRollOnOff: R_TRIG;
	fbCountBtwUnwindPulse: CTU;

	bIgnoreFirstUnwindPulse: BOOL;
	iCountBtwUnwindPulseLatched: INT:= 30;
	fbRTrigUnwind: R_TRIG;
	fbFTrigUnwind: F_TRIG;
	iCountBtwUnwindPulseLimit: INT := 15;
	rMyMod: DINT;
	rMyPosition: REAL;
	diMyPosition: DINT;
	diMyReference: DINT;
	diMasterPos: DINT;
	diOffset: DINT;
	bFlag: BOOL;
	//fbBlink: BLINK;
	rActualSpeed: REAL;
	tPeriodTime: TIME;
	tTimeOff: TIME;
	rPeriodTime: REAL;
	tPeriod: TIME;
	rTimeOff: REAL;
	diActualSpeed: DINT;
	tTimeQuelconque: TIME;
	TPInst: TP;
	tTimeOn: TIME;
	rTimeOn: REAL;
	diLastSetpoint: DINT;
	diCurrentSpeedsetpoint: DINT;
//	fbHysteresis: HYSTERESIS;
	rEffectiveRepeat: REAL;
	bEnableBogus: BOOL;


	(*FOR UNWIND*)
	uiStep: UINT;
	fbFiltPulse: IL_StatisticType01;
	ComputeOn: BOOL;
	StatOn: BOOL;
	StatError: BOOL;
	StatErrorStruct: ERROR_STRUCT;
	StatErrorID: ERROR_CODE;
	StatPaused: BOOL;
	rPulseMean_gb: REAL;
	rPulseVariance_gb: REAL;
	rStartDiam: REAL := 100000;
	rDiamMean_gb: REAL;
//	fbDiamRamp: RAMP_REAL;
	rDiamFinal_gb: REAL;

	rMinValue: REAL;
	rMaxValue: REAL;
	bResetCTU: BOOL;

	bWinder1OffSw_q: BOOL;
	bWinder2OffSw_q: BOOL;
	bRewindCalculationEnable: BOOL;
	bRewindCalculationMinTensAchieved: BOOL;
	rUnwindTensCtrl_HighHysteresisLimit: REAL;
	rUnwindTensCtrl_LowHysteresisLimit: REAL;
//	fbMinTens_UnwindDiamCalcEnable: HYSTERESIS;
	uiUnwindTensCtrl_LowHysteresisLimit: UINT;
	uiUnwindTensCtrl_HighHysteresisLimit: UINT;
	uiUnwindTensCtrl_ScaledFBK_HMI: UINT;
	uiUnwindTensCtrl_ScaledFBK: UINT;
	bUnwindCalculationMinTensAchieved: BOOL;
	df: BOOL;
	bNOTUnwindCalculationMinTensAchieved: BOOL;

	fbCatchDiam: F_TRIG;
	bMinSpeedAchieved: BOOL;
	fbNewRoll: TP;
	bNewRoll_Unwind_Seq: BOOL;

	rSetpointInNewtonsW1: REAL;
	rSetpointInNewtonsW2: REAL;

	rCurrentDiameterW1_buff: REAL;
	fb_ResetEND_OF_ROLL_ACTIVE: R_TRIG;
	
	bResetFirstUnwindPulse: BOOL := FALSE;
	fbFirstUnwindPulse: CTU;
	uiFirstUnwindCount: UINT;
	fbFirstWebBreakPulse: CTU;
	fbEndOfRollOnOff_WB: R_TRIG;
	uiFirstUnwindCount_WB: UINT;
	bIgnoreFirstUnwindPulse_WB: BOOL;
	fbCountBtwUnwindPulse_WB: CTU;
	iCountBtwUnwindPulse_WB: INT;
	fbWebBreakOnOff: R_TRIG;
END_VAR



VAR_INPUT


	bWinder1Direction		: BOOL;
	bWinder2Direction		: BOOL;
	rRepeat_i				: REAL;

END_VAR

VAR CONSTANT



	COREVAL_3INCH:			REAL:= 76.2;
	COREVAL_6INCH:			REAL:= 160.0;
	MAXDIAMETER:			REAL:= 508.0;		(* Arbitrary Value for this *)
	MINDIAMETER: 			REAL:= 76.2;
	MECHINERTIA_3INCH:		REAL:= 0.005137; 	(* Arbitrary, follow procedure to calculate Inertia *)
	MECHINERTIA_6INCH:		REAL:= 0.0475;
	MECHINERTIA:			REAL:= 0.005137;
	STANDSTILLTORQUE:		REAL:= 3.0;		(* Original value 3.0  *)	(* Arbitrary, follow procedure to evaluate torque *)
	MINTORQUE :				REAL:= 3.0;		(* Original value 3.0  *)
	MINTORQUEVELOCITY:		REAL:= 5; 	(* Original value 10.0  *)(* RPM *)
	MAXTORQUE:				REAL:= 6.0;		(* Original value 7.0  *)(* % At S91*)
	MOTORMAXTORQUE: 		REAL:= 12500.0; (* NewtonMilliMeters *)
	MINTENSION:				REAL:= 5.0;	(* Newtons *)
	ANALOG_SCALING_W1:		REAL:= 10.0;
	ANALOG_SCALING_W2:		REAL:= 10.0;
	MINWEBWIDTH:			REAL:= 25.4;  (* arbitrary Min value *)



	iCountPerBatch12: 				INT := 12;
	rOneMeter_In_Inches: 	REAL := 39.37;	(*INCHES*)

	rPI	: 					REAL := 3.14159;
	diCountMargin : 		DINT := 5;

END_VAR

(* time measurement *)
LowTimeTickWindTens := ( IL_HighResTimeTick (TRUE) );


	//rTensionSpeedW1 := UINT_TO_REAL( (10.0 * 10000) / (uiFormat_gb));


	(*- - - WINDER #1 - - -*)

	(* A - Diameter Setup *)

	stWindTensDiamW1.CoreVal			:= 90.0;			(* 83mm *)
	stWindTensDiamW1.Density			:= rDensity;		(* 0.771 kg/dm^3 *)
	stWindTensDiamW1.MaxDiameter		:= MAXDIAMETER;		(* 508mm - 20 inches*)
	stWindTensDiamW1.MinDiameter		:= MINDIAMETER;
	stWindTensDiamW1.MechanicInertia	:= MECHINERTIA_3INCH;
	stWindTensDiamW1.RepeatLength		:= 100.0;
	stWindTensDiamW1.PresetVal			:= rStartDiameterW1_HMI * 25.4;
	stWindTensDiamW1.WebWidth			:= rWebWidthRew1;	(* 407mm*)
	stWindTensDiamW1.AverageValue		:= iDiameterAvg;
	stWindTensDiamW1.LowLimit			:=	MINDIAMETER;
	stWindTensDiamW1.HighLimit			:=	MAXDIAMETER;
	stWindTensDiamW1.DiamCalcMode		:=   CALC_DIAM_MANUAL(*FIRST_REV_AUTO_CALC*);

	(* B - Friction Setup *)

    stWindFrictionW1.MaxTorque			:= MAXTORQUE;
	stWindFrictionW1.MinTorque			:= MINTORQUE;
	stWindFrictionW1.StandstillTorque	:= STANDSTILLTORQUE;
	stWindFrictionW1.MinTorqueVelocity	:= MINTORQUEVELOCITY;

	(* WINDER #1,  WITHOUT VISUALIZATION *)

    fbWindTension_W1(
		Enable:=TRUE ,
		Pause:= bPauseW1 ,
		DisableCyclicWrites := FALSE,
		WindCtrlType		:= OPEN_LOOP,
		WindDirection		:= REWIND,
		PauseDiameter		:=  FALSE,
		PresetDiameter		:= (bNewRoll_Winder1_HMI_i OR bFirstPresetW1) ,
		TensionMode			:= CONST_WEB_VEL,
		SetpointStandstill	:= rWinder1_Standstill_TensionHMI_gb * 4.4,//multiply by 4.4 to get in lbs.
		SetpointOpMode		:= rTensionSetpointW1_HMI_i *4.4,
		TensionSpeed		:= rTensionSpeedW1 ,
		ActTorqueFilter		:= tActualTorqFilterW1 ,
		AccelTorqueFilter	:= tAccelTorqFilterW1 ,
		DefaultTorqueLimit	:= rDefTorqueLimW1 ,
        WindowTension		:= rWindowInTensionPctW1,
        MinTension			:= rMinTensionMonitorW1,
        MaxTension			:= rMaxTensionMonitorW1 ,
		Diameter			:= stWindTensDiamW1,     (* Diameter Structure *)
		TensionCtrl			:= stWindTensionCtrlW1 , (* Tension Control Structure only with Load cell.*)
		Friction			:= stWindFrictionW1,     (* Structure for Friction *)
		Master				:= VMA_FT1,(*Axis3,VmAxisExt,*)
		Slave				:= arAxisCtrl_gb[Drive20.AxisNo].Admin.Axis,
		InOperation 		=> bInOperationW1,
		Error 				=> bErrorW1,
		ErrorID=> ,
		ErrorIdent			=> stErrorIdentW1,
		InPause				=> bInPauseW1,
		PresetDiamAck		=> bPresetDiamAckW1,
		InPauseDiam			=> bInPauseDiamW1,
		MinAvDiamAchieved	=> bMinAvDiamAchievedW1,
		MaxAvDiamAchieved	=> bMaxAvDiamAchievedW1,
		HighLimitDiamActive	=> bHighLimitDiamActiveW1,
		LowLimitDiamActive	=> bLowLimitDiamActiveW1,
        TensionInWindow		=> bTensionInWindowW1,
        MinTensionAchieved	=> bMinTensionAchievedW1,
        MaxTensionAchieved	=> bMaxTensionAchievedW1,
	    DiameterEngaged		=> bDiameterEngagedW1,
	    HighLimitTensActive	=> bHighLimitTensActiveW1,
	    LowLimitTensActive	=> bLowLimitTensActiveW1,
		CurrentDiameter		=> 	rCurrentDiameterW1,
		GearRatioFineAdjust	=> 	rGearRatioFineAdjustW1,
		CurrentInertia		=> 	rCurrentInertiaW1,
		SpeedOffset			=> 	rSpeedOffsetW1,
		TorqueLimitBipolar	=> 	rTorqueLimitBipolarW1,
		WindTensDiag		=> 	stWindTensDiagW1);


		rGearRatioFineAdjustW1_HMI	:= rGearRatioFineAdjustW1;
		rSpeedOffsetW1_HMI			:= rSpeedOffsetW1;
		rCurrentDiameterW1_HMI		:=	rCurrentDiameterW1/ 25.4;
		//rCurrentDiameterW1_HMI		:=	rCurrentDiameterW1;


		(*THE BLOODY BUTTON GOT STUCK-> QUICK FIX*)
		IF fbWindTension_W1.PresetDiamAck THEN
			bFirstPresetW1:= FALSE;
		END_IF

	(*- - - WINDER #2 - - -*)
	(*rTensionSpeedW2 := (10.0 * 10000) / (uiFormat_gb);
	(* A - Diameter Setup *)

	stWindTensDiamW2.CoreVal			:= rCoreSize_gb;
	stWindTensDiamW2.Density			:= rDensity;
	stWindTensDiamW2.MaxDiameter		:= MAXDIAMETER;
	stWindTensDiamW2.MinDiameter		:= MINDIAMETER;
	stWindTensDiamW2.MechanicInertia	:= rMechInertia_gb;
	stWindTensDiamW2.RepeatLength		:= rFormat_gb;
	stWindTensDiamW2.PresetVal			:= rStartDiameterW2_HMI * 25.4;
	stWindTensDiamW2.WebWidth			:= rWebWidthRew2;

	stWindTensDiamW2.DiamCalcMode		:= FIRST_REV_AUTO_CALC;
	stWindTensDiamW2.LowLimit			:=	MINDIAMETER;
	stWindTensDiamW2.HighLimit			:=	MAXDIAMETER;

	(* B - Friction Setup *)

    stWindFrictionW2.MaxTorque			:= MAXTORQUE;
	stWindFrictionW2.MinTorque			:= MINTORQUE;
	stWindFrictionW2.StandstillTorque	:= STANDSTILLTORQUE;
	stWindFrictionW2.MinTorqueVelocity	:= MINTORQUEVELOCITY;

	 fbWindTension_W2(
		Enable				:=bEnableW2 OR bEnableBogus ,
		Pause				:=  bPauseW2 ,
		DisableCyclicWrites := FALSE ,
		WindCtrlType		:= OPEN_LOOP,
		WindDirection		:= REWIND,
		PauseDiameter		:= bManAutoTensionControl_i,
		PresetDiameter		:= (bNewRoll_Winder2_HMI_i OR bFirstPresetW2) (* OR bPresetDebuggerW2)*) AND Prog_Operating_Modes.stpStoppedAndPulling.x AND arAxisStatus[3].Admin.MODE_AH,
		TensionMode			:= CONST_WEB_VEL,
		SetpointStandstill	:= rWinder1_Standstill_TensionHMI_gb * 4.4,
		SetpointOpMode		:= rSetPointProcessedW2,
		TensionSpeed		:= rTensionSpeedW2  ,
		ActTorqueFilter		:= tActualTorqFilterW2,
		AccelTorqueFilter	:= tAccelTorqFilterW2,
		DefaultTorqueLimit	:= rDefTorqueLimW2,
  		WindowTension		:= rWindowInTensionPctW2,
        MinTension			:= rMinTensionMonitorW2,
        MaxTension			:= rMaxTensionMonitorW2,
		Diameter			:= stWindTensDiamW2,     (* Diameter Structure *)
		TensionCtrl			:= stWindTensionCtrlW2 , (* Tension Control Structure only with Load cell.*)
		Friction			:= stWindFrictionW2,     (* Structure for Friction *)
		Master				:= VmAxisExt,
		Slave				:= Axis2,
		InOperation 		=> bInOperationW2,
		Error 				=> bErrorW2,
		ErrorID=> ,
		ErrorIdent			=> stErrorIdentW2,
		InPause				=> bInPauseW2,
		PresetDiamAck		=> bPresetDiamAckW2,
		InPauseDiam			=> bInPauseDiamW2,
		MinAvDiamAchieved	=> bMinAvDiamAchievedW2,
		MaxAvDiamAchieved	=> bMaxAvDiamAchievedW2,
		HighLimitDiamActive	=> bHighLimitDiamActiveW2,
		LowLimitDiamActive	=> bLowLimitDiamActiveW2,
        TensionInWindow		=> bTensionInWindowW2,
        MinTensionAchieved	=> bMinTensionAchievedW2,
        MaxTensionAchieved	=> bMaxTensionAchievedW2,
	    DiameterEngaged		=> bDiameterEngagedW2,
	    HighLimitTensActive	=> bHighLimitTensActiveW2,
	    LowLimitTensActive	=> bLowLimitTensActiveW2,
		CurrentDiameter		=> rCurrentDiameterW2,
		GearRatioFineAdjust	=> rGearRatioFineAdjustW2,
		CurrentInertia		=> rCurrentInertiaW2,
		SpeedOffset			=> rSpeedOffsetW2,
		TorqueLimitBipolar	=> rTorqueLimitBipolarW2,
		WindTensDiag		=> stWindTensDiagW2);

		rGearRatioFineAdjustW2_HMI	:= rGearRatioFineAdjustW2;
		rSpeedOffsetW2_HMI			:= rSpeedOffsetW2;
		(*rCurrentDiameterW2_HMI		:=	rCurrentDiameterW2/ 25.4;*)
		rCurrentDiameterW2_HMI		:=	rCurrentDiameterW2;


		(*THE BLOODY BUTTON GOT STUCK-> QUICK FIX*)
		IF bPresetDiamAckW2=TRUE THEN

			bNewRoll_Winder2_HMI_i := FALSE;

		END_IF*)


(* time measurement *)
 HighTimeTickWindTens := ( IL_HighResTimeTick (TRUE) );

 TimeDiffWindTens := IL_HighResTimeDiff ( LowTimeTickWindTens, HighTimeTickWindTens );
 TimeMaxWindTens := MAX (TimeDiffWindTens, TimeMaxWindTens);

END_PROGRAM

// IndraMotionMlc1/Application/AxisInterface/_Readme
PROGRAM _Readme
VAR
END_VAR

;
(*  English                              | Deutsch
Please do not change the programs and    | Bitte die Programme und Funktionsbausteine
function blocks in this folder. Updates  | in diesem Ordner nicht veraendern. Updates des
of the AxisInterface example project     | AxisInterface Besipielprojektes werden eine
will include an EXPORT-File with the     | EXPORT-Datei mit dem Inhalt dieses Ordners enthalten.
content of this folder.                  |
If you want to adapt the POUs, copy and  | Bei Anpassungen an den POEs bitte kopieren und 
rename it to avoid overwriting           | umbenennen, um ein Ueberschreiben zu vermeiden  *)

END_PROGRAM

// IndraMotionMlc1/Application/Utilities/AllAxisAB
PROGRAM AllAxisAB
VAR_INPUT
	arAxisPointer: POINTER TO ARRAY[1..20] OF AXIS_REF;
	uiNUM_FLEXO_F: UINT;
END_VAR
VAR_OUTPUT
	
	bAllAxisHealthy:BOOL;
END_VAR
VAR
	index : UINT :=1;
END_VAR

bAllAxisHealthy := TRUE;

FOR index:=1 TO uiNUM_FLEXO_F BY 1 DO
	IF 	arAxisStatus_gb[arDrive[index].AxisNo].Admin._OpModeAck=ModeAB THEN
		;//do nothing (it stays true)
	ELSE
		bAllAxisAB := FALSE;
	END_IF
END_FOR

END_PROGRAM

// IndraMotionMlc1/Application/Utilities/UnSynchronizePullroll
PROGRAM UnSynchronizePullroll
VAR
END_VAR

END_PROGRAM

// IndraMotionMlc1/Application/Expectation Window Managment/ML_RegiCtrlExpectWinType01/ML_RegiCtrlExpectWinType01

(*#############################################################################################
  #############################################################################################  

   General Header   
  ---------------------------------------------------------------------------------------------  
   Shortdescription       : Handles the Probe expectation windows when Register Controller are started
   Version                :  2T00
   Name                   : DCCA/GB
   Date                   :  Nov 15Th, 2011 , Jan 2014, July 2014
   Company                : Bosch Rexroth Canada Inc.  
   Target                 : IndraMotion MLC 11/12/13
   Functional description : In conjunction with a register Controller signals, Opens up and Close Probe Expectation Windows and deliver Done signal for Regulator
   							The Windows Setpoint given by The Register controller.
   
   
   
   
   
 
   Handling specials      : 							
						 
  ---------------------------------------------------------------------------------------------  
    
   Modification and History :
   
   *)

FUNCTION_BLOCK ML_RegiCtrlExpectWinType01



VAR_INPUT
	Enable:BOOL;
	RegisterInOperation:BOOL;
	SetPointLockAck:BOOL;
	SetPoint:REAL;
	Incr:BOOL;
	ExpectWindowPosLimit:LREAL;
	ExpectWindowNegLimit:LREAL;
	
	
	
	
	
	
	
	

END_VAR



VAR_OUTPUT
	InOperation:BOOL;
	Done:BOOL;
	StorageModeCmd:UINT;
	StorageCmdExe:BOOL;
	Error:BOOL;
	ErrorID:ERROR_CODE ;
	ErrorIdent: ERROR_STRUCT;

END_VAR



VAR
	
	enState: ML_REGICTRL_EXPECTWIN_TYPE01;
	cnt:int;
	bExeExpectWin: BOOL;
	bExeWindowsDone: BOOL;
	fbStorageMode: MB_WriteParameter;
	bRuntime_Busy:BOOL;
	
	fbWriteExpectWindow: ML_WriteExpectWinPosEdgeType01;
	uiShutDownState: INT;
	strErrorSource: STRING(INT#16);
	bStorageModeDone: BOOL;
END_VAR




VAR_IN_OUT
 Axis:AXIS_REF;
 
END_VAR

VAR CONSTANT

MAXPOSLIMITDEG:REAL:=179.9;(* Maximum value for Positive limit of Expextation Window*)
MINNEGLIMITDEG:REAL:=179.9; (* Minimum value for Negative limit of Expextation Window*)

MAXPOSLIMITINCR:REAL:=524288;(* Maximum value for Positive limit of Expextation Window*)
MINNEGLIMITINCR:REAL:=524287; (* Minimum value for Negative limit of Expextation Window*)


END_VAR




	IF ( Enable AND enState = ML_REGICTRL_EXPECTWIN_TYPE01.STATE_IDLE)  THEN 
		enState:= ML_REGICTRL_EXPECTWIN_TYPE01.STATE_STORAGE_MODE_OFF ;
	END_IF
	
	
	IF  ( NOT Enable AND bRuntime_Busy ) THEN
		enState:= ML_REGICTRL_EXPECTWIN_TYPE01.STATE_SHUTDOWN ;
	END_IF

	
	InOperation:= enstate <> ML_REGICTRL_EXPECTWIN_TYPE01.STATE_IDLE AND NOT ERROR;
	
	
	
	
	
	CASE enState OF 
		
	
		ML_REGICTRL_EXPECTWIN_TYPE01.STATE_IDLE:

		
			(*Do nothing*);
						
		
			
		ML_REGICTRL_EXPECTWIN_TYPE01.STATE_STORAGE_MODE_OFF:(*Drive Flash Storage must be Off*)
			
			
			bExeWindowsDone:=FALSE;
			uiShutDownState:=0;
			bRuntime_Busy:=TRUE;
			StorageModeCmd:=1;
			StorageCmdExe:=TRUE;
			
			enState:=ML_REGICTRL_EXPECTWIN_TYPE01.STATE_WAIT_REGI_IN_OPERATION;
	
		
				
		ML_REGICTRL_EXPECTWIN_TYPE01.STATE_WAIT_REGI_IN_OPERATION:
				
			
			
			//Open Windows:
			
			IF Incr THEN	
				
											
				fbWriteExpectWindow(
					Execute:= TRUE, 
					SetPoint:=0 , 
					Incr:=Incr,
					ExpectWindowPosLimit:=MAXPOSLIMITINCR , 
					ExpectWindowNegLimit:=MINNEGLIMITINCR , 
					Axis:=Axis , 
					Done=>, 
					Error=> , 
					ErrorID=> , 
					ErrorIdent=> );
			ELSE
			
									
				fbWriteExpectWindow(
					Execute:= TRUE, 
					SetPoint:=180.0 ,
					Incr:=Incr, 
					ExpectWindowPosLimit:=MAXPOSLIMITDEG , 
					ExpectWindowNegLimit:=MINNEGLIMITDEG , 
					Axis:=Axis , 
					Done=> , 
					Error=> , 
					ErrorID=> , 
					ErrorIdent=> );

			END_IF
			
			
			
						
			IF fbWriteExpectWindow.Done THEN
				
				enState:= ML_REGICTRL_EXPECTWIN_TYPE01.STATE_RESET_FB_INST;
				
			ELSIF fbWriteExpectWindow.Error THEN
			
				ErrorIdent:= fbWriteExpectWindow.ErrorIdent;
				ErrorID:=fbWriteExpectWindow.ErrorID;
				enState:=ML_REGICTRL_EXPECTWIN_TYPE01.STATE_ERROR;
				
			END_IF
	
				
		
		ML_REGICTRL_EXPECTWIN_TYPE01.STATE_RESET_FB_INST:
		
		
				//Reset Expect Window Instance												
				fbWriteExpectWindow(
					Execute:= FALSE, 
					SetPoint:=0 , 
					Incr:=Incr,
					ExpectWindowPosLimit:=MAXPOSLIMITINCR , 
					ExpectWindowNegLimit:=MINNEGLIMITINCR , 
					Axis:=Axis , 
					Done=>, 
					Error=> , 
					ErrorID=> , 
					ErrorIdent=> );
					
					
				enState:=ML_REGICTRL_EXPECTWIN_TYPE01.STATE_WAIT_REGI_SETPOINT_LOCK;
		
				
				
		
				
		ML_REGICTRL_EXPECTWIN_TYPE01.STATE_WAIT_REGI_SETPOINT_LOCK: // WAIT FOR SETPOINT LOCKED
			
		
			//Close Windows around SetPoint	
			
			IF ( SetPointLockAck AND RegisterInOperation) THEN
			
						
								
			fbWriteExpectWindow(
				Execute:= TRUE, 
				SetPoint:=Setpoint , 
				ExpectWindowPosLimit:=ExpectWindowPosLimit , 
				ExpectWindowNegLimit:=ExpectWindowNegLimit , 
				Axis:=Axis , 
				Done=> , 
				Error=> , 
				ErrorID=> , 
				ErrorIdent=> );		


			
		
			(*   Embedded ML_WriteEpexctWinPosEdgeType01   *)
			
			IF fbWriteExpectWindow.Done THEN
				
				Done:=TRUE;
				enState:=ML_REGICTRL_EXPECTWIN_TYPE01.STATE_RUN;
				
			ELSIF fbWriteExpectWindow.Error THEN
			
				ErrorIdent:= fbWriteExpectWindow.ErrorIdent;
				ErrorID:=fbWriteExpectWindow.ErrorID;
				enState:= ML_REGICTRL_EXPECTWIN_TYPE01.STATE_ERROR;
				
			END_IF
			

	
							
		END_IF		
			
			
					
		ML_REGICTRL_EXPECTWIN_TYPE01.STATE_RUN:// RUN
		
			StorageCmdExe:=FALSE;

			//Reset Fb instance from actCloseWindows									
			fbWriteExpectWindow(
				Execute:= FALSE, 
				SetPoint:=Setpoint ,
				Incr:=Incr, 
				ExpectWindowPosLimit:=ExpectWindowPosLimit , 
				ExpectWindowNegLimit:=ExpectWindowNegLimit , 
				Axis:=Axis , 
				Done=> , 
				Error=> , 
				ErrorID=> , 
				ErrorIdent=> );
					;
					
					
					
		
			// Re-Run Conditions:		
			IF ( RegisterInOperation AND NOT SetPointLockAck  ) OR  ( NOT RegisterInOperation ) THEN
				Done:=FALSE;
				enState:=ML_REGICTRL_EXPECTWIN_TYPE01.STATE_WAIT_REGI_IN_OPERATION;
			END_IF
		
					
			
		ML_REGICTRL_EXPECTWIN_TYPE01.STATE_SHUTDOWN:

		
			actShutdown();
		
			
		ML_REGICTRL_EXPECTWIN_TYPE01.STATE_ERROR:
			

			Error:=TRUE;
	
				
					
		ML_REGICTRL_EXPECTWIN_TYPE01.STATE_DUMMY:
		;
	
	END_CASE

ACTION actShutdown:
(*Action Shutdown*)


	CASE uiShutDownState OF
	
		0:// Close fbWriteExpectWindow
		
	
		fbWriteExpectWindow(
			Execute:= FALSE, 
			SetPoint:=Setpoint ,
			Incr:=Incr, 
			ExpectWindowPosLimit:=ExpectWindowPosLimit , 
			ExpectWindowNegLimit:=ExpectWindowNegLimit , 
			Axis:=Axis , 
			Done=> , 
			Error=> , 
			ErrorID=> , 
			ErrorIdent=> );
				;
			StorageCmdExe:=FALSE;
			uiShutDownState:=10;
				
		10://Turn off Storage Mode	
		
		
			StorageModeCmd:=0;
			StorageCmdExe:=TRUE;
			uiShutDownState:=20;
			
		20:// Turn Off Commands
		
					
			StorageCmdExe:=FALSE;	
			bRuntime_Busy:=FALSE;
			Error:=FALSE;
			Done:=FALSE;
			
			enState:= ML_REGICTRL_EXPECTWIN_TYPE01.STATE_IDLE;
		
			
	END_CASE
END_ACTION

END_FUNCTION_BLOCK

// IndraMotionMlc1/Application/Expectation Window Managment/ML_WriteExpectWinPosEdgeType01/ML_WriteExpectWinPosEdgeType01
FUNCTION_BLOCK ML_WriteExpectWinPosEdgeType01
(*#############################################################################################
  #############################################################################################  

   General Header   
  ---------------------------------------------------------------------------------------------  
   Shortdescription       : Write Expecation WIndows   Version                :  2T00
   Name                   : DCCA/GB
   Date                   :  July 2014
   Company                : Bosch Rexroth Canada Inc.  
   Target                 : IndraMotion MLC 11/12/13
   Functional description : write expectation Windows, Degrees or Increments
   
   
   
   
   
 
   Handling specials      : 	Call in PLC program, avoid Motion Task since this fb use acylcic transmission of -Parameters
								Turn off Storage Mode of Drive, parameter S-0-0269 to avoid damage to flash memory						
						 
  ---------------------------------------------------------------------------------------------  
    
   Modification and History :
   
   25/07/2014 : added Type of Axis : Distinction bewtween Inc and Degrees
   
   *)
   
VAR_INPUT
	Execute:BOOL;
	SetPoint:REAL;
	Incr:BOOL;		(*If True then the windows are calculated in increment 2^20 incr *)
	ExpectWindowPosLimit:LREAL;
	ExpectWindowNegLimit:LREAL;
	
END_VAR
VAR_OUTPUT
	Done:BOOL;
	Error:BOOL;
	ErrorID:ERROR_CODE ;
	ErrorIdent: ERROR_STRUCT;
END_VAR
VAR
	enState: ML_WRITE_EXPECT_WIN_TYPE01;
	bOldExecute: BOOL;
	rP204StartPos: REAL;
	diP204StartPos:DINT;
	diP205EndPos:DINT;	
	rP205EndPos: REAL;
	fbWriteParam: MB_WriteRealParameter;
	fbWriteParamDint: MB_WriteParameter;
		
END_VAR
VAR_IN_OUT
	Axis:Axis_Ref;
	
END_VAR




IF Execute AND NOT bOldExecute THEN
	enState:= ML_WRITE_EXPECT_WIN_TYPE01.STATE_CHECK_VALIDITY;
END_IF

IF NOT Execute AND  ( enState<> ML_WRITE_EXPECT_WIN_TYPE01.STATE_SHUTDOWN ) THEN
enState:= ML_WRITE_EXPECT_WIN_TYPE01.STATE_SHUTDOWN;
END_IF


//Main



	CASE enState OF
		
	
	
		ML_WRITE_EXPECT_WIN_TYPE01.STATE_IDLE:
		
			RETURN;
		
		
		ML_WRITE_EXPECT_WIN_TYPE01.STATE_CHECK_VALIDITY:
		
		
			IF Incr THEN
				
				IF  ( ExpectWindowPosLimit > 1048576  OR 	ExpectWindowNegLimit < 0 ) THEN
					Error:= TRUE;
					ErrorIdent.Table:=F_RELATED_TABLE;
					ErrorIdent.Additional1:=16#00000002;
					ErrorID:=INPUT_RANGE_ERROR;
					enState:= ML_WRITE_EXPECT_WIN_TYPE01.STATE_ERROR ;
					
				ELSE
					enState:=ML_WRITE_EXPECT_WIN_TYPE01.STATE_CALC_WINDOWS;
			
				END_IF
			
			
			
			ELSE
			
					IF  ( ExpectWindowPosLimit > 180.0  OR 	ExpectWindowNegLimit > 180.0 ) THEN
						Error:= TRUE;
						ErrorIdent.Table:=F_RELATED_TABLE;
						ErrorIdent.Additional1:=16#00000002;
						ErrorID:=INPUT_RANGE_ERROR;
						enState:= ML_WRITE_EXPECT_WIN_TYPE01.STATE_ERROR ;
						
					ELSE
						enState:=ML_WRITE_EXPECT_WIN_TYPE01.STATE_CALC_WINDOWS;
				
					END_IF
					
			END_IF
				
			
		ML_WRITE_EXPECT_WIN_TYPE01.STATE_CALC_WINDOWS:


		IF Incr THEN
				
									
				//(*Caclulates Windows Modulo 1048576 incr*)
				rP204StartPos	:=	MB_GetModuloType01(Value:= SetPoint - ExpectWindowNegLimit ,  ModuloValue:= 1048576 );
				rP205EndPos	:=  MB_GetModuloType01(Value:= ExpectWindowPosLimit + SetPoint    ,   ModuloValue:= 1048576);
				
				diP204StartPos:=REAL_TO_DINT(rP204StartPos);
				diP205EndPos:=REAL_TO_DINT(rP205EndPos);
				
				enState:= ML_WRITE_EXPECT_WIN_TYPE01.STATE_WRITE_START_POS;
				
			
			ELSE
			
				
				(*Caclulates Windows Modulo 360.0 degres*)
				rP204StartPos 	:=	MB_GetModuloType01(Value:= SetPoint  -  ExpectWindowNegLimit ,  ModuloValue:= 360.0 );
				rP205EndPos	:=  MB_GetModuloType01(Value:= ExpectWindowPosLimit + SetPoint    ,   ModuloValue:= 360.0);
				
				enState:= ML_WRITE_EXPECT_WIN_TYPE01.STATE_WRITE_START_POS;
			
			END_IF
			
			
			 
		ML_WRITE_EXPECT_WIN_TYPE01.STATE_WRITE_START_POS:(*Negative Limit*)
		
			
		
				IF Incr THEN
		
					fbWriteParamDint(
						Execute:=TRUE , 
						ParameterNumber:=GVL_P_Param_ID.FP_P_0_0204 , 
						Value:=diP204StartPos , 
						Axis:=Axis, 
						Done=> , 
						Active=> , 
						Error=> , 
						ErrorID=> , 
						ErrorIdent=> );
						
						
						IF  fbWriteParamDint.Done THEN 
						enState:=ML_WRITE_EXPECT_WIN_TYPE01.STATE_RESET_PARAM_INST;
				 	ELSIF	fbWriteParam.Error THEN
						ErrorID:=  fbWriteParamDint.ErrorID;
						ErrorIdent :=fbWriteParamDint.ErrorIdent;
						enState:= ML_WRITE_EXPECT_WIN_TYPE01.STATE_ERROR;
					END_IF
					
				
				ELSE
				
					fbWriteParam(
						Execute:= TRUE, 
						ParameterNumber:= GVL_P_Param_ID.FP_P_0_0204 , 
						Value:=rP204StartPos , 
						Axis:=Axis , 
						Done=> , 
						Active=> , 
						Error=> , 
						ErrorID=> , 
						ErrorIdent=> );
						
						
						
					IF  fbWriteParam.Done THEN 
						enState:=ML_WRITE_EXPECT_WIN_TYPE01.STATE_RESET_PARAM_INST;
				 	ELSIF	fbWriteParam.Error THEN
						ErrorID:=  fbWriteParam.ErrorID;
						ErrorIdent :=fbWriteParam.ErrorIdent;
						enState:= ML_WRITE_EXPECT_WIN_TYPE01.STATE_ERROR;
					END_IF
						
					
				END_IF
									
			
				
				
		ML_WRITE_EXPECT_WIN_TYPE01.STATE_RESET_PARAM_INST:

			fbWriteParam(
				Execute:= FALSE, 
				Axis:=Axis , 
					 	);
			
			fbWriteParamDint(
				Execute:=FALSE , 
				ParameterNumber:=GVL_P_Param_ID.FP_P_0_0204 , 
				Value:=diP204StartPos , 
				Axis:=Axis, 
				Done=> , 
				Active=> , 
				Error=> , 
				ErrorID=> , 
				ErrorIdent=> );
						
					
				enState:= ML_WRITE_EXPECT_WIN_TYPE01.STATE_WRITE_END_POS;	
				
				

		ML_WRITE_EXPECT_WIN_TYPE01.STATE_WRITE_END_POS:(*Positive Limit*)
			
		
		
		
			IF Incr THEN // a DINT is written
			
				fbWriteParamDint(
					Execute:=TRUE , 
					ParameterNumber:=GVL_P_Param_ID.FP_P_0_0205 , 
					Value:=diP205EndPos , 
					Axis:=Axis, 
					Done=> , 
					Active=> , 
					Error=> , 
					ErrorID=> , 
					ErrorIdent=> );
						
					
